      movel(pose_trans(ref_frame,p[0.079719, 0.078170, -0.000125, -0.013708, 3.141563, -0.000000]),accel_mss,speed_ms,0,0.001)
      movel(pose_trans(ref_frame,p[0.079740, 0.078322, -0.000125, -0.013708, 3.141563, 0.000000]),accel_mss,speed_ms,0,0.001)
      movel(pose_trans(ref_frame,p[0.079758, 0.078475, -0.000125, -0.013708, 3.141563, -0.000000]),accel_mss,speed_ms,0,0.001)
      movel(pose_trans(ref_frame,p[0.079771, 0.078603, -0.000125, -0.013708, 3.141563, 0.000000]),accel_mss,speed_ms,0,0.001)
      movel(pose_trans(ref_frame,p[0.079782, 0.078732, -0.000125, -0.013708, 3.141563, 0.000000]),accel_mss,speed_ms,0,0.001)
      movel(pose_trans(ref_frame,p[0.079779, 0.078758, -0.000125, -0.013708, 3.141563, 0.000000]),accel_mss,speed_ms,0,0.001)
      movel(pose_trans(ref_frame,p[0.079765, 0.078781, -0.000125, -0.013708, 3.141563, 0.000000]),accel_mss,speed_ms,0,0.001)
      movel(pose_trans(ref_frame,p[0.079742, 0.078796, -0.000125, -0.013708, 3.141563, 0.000000]),accel_mss,speed_ms,0,0.001)
      movel(pose_trans(ref_frame,p[0.079715, 0.078802, -0.000125, -0.013708, 3.141563, 0.000000]),accel_mss,speed_ms,0,0.001)
      movel(pose_trans(ref_frame,p[0.079591, 0.078803, -0.000125, -0.013708, 3.141563, 0.000000]),accel_mss,speed_ms,0,0.001)
      movel(pose_trans(ref_frame,p[0.079467, 0.078802, -0.000125, -0.013708, 3.141563, 0.000000]),accel_mss,speed_ms,0,0.001)
      movel(pose_trans(ref_frame,p[0.079319, 0.078800, -0.000125, -0.013708, 3.141563, -0.000000]),accel_mss,speed_ms,0,0.001)
      movel(pose_trans(ref_frame,p[0.079172, 0.078794, -0.000125, -0.013708, 3.141563, 0.000000]),accel_mss,speed_ms,0,0.001)
      movel(pose_trans(ref_frame,p[0.079002, 0.078785, -0.000125, -0.013708, 3.141563, 0.000000]),accel_mss,speed_ms,0,0.001)
      movel(pose_trans(ref_frame,p[0.078832, 0.078774, -0.000125, -0.013708, 3.141563, -0.000000]),accel_mss,speed_ms,0,0.001)
      movel(pose_trans(ref_frame,p[0.077770, 0.078748, -0.000125, -0.013708, 3.141563, -0.000000]),accel_mss,speed_ms,0,0.001)
      movel(pose_trans(ref_frame,p[0.076711, 0.078827, -0.000125, -0.013708, 3.141563, 0.000000]),accel_mss,speed_ms,0,0.001)
      movel(pose_trans(ref_frame,p[0.075653, 0.079010, -0.000125, -0.013708, 3.141563, -0.000000]),accel_mss,speed_ms,0,0.001)
      movel(pose_trans(ref_frame,p[0.074616, 0.079292, -0.000125, -0.013708, 3.141563, -0.000000]),accel_mss,speed_ms,0,0.001)
      movel(pose_trans(ref_frame,p[0.073606, 0.079674, -0.000125, -0.013708, 3.141563, 0.000000]),accel_mss,speed_ms,0,0.001)
      movel(pose_trans(ref_frame,p[0.072636, 0.080148, -0.000125, -0.013708, 3.141563, 0.000000]),accel_mss,speed_ms,0,0.001)
      movel(pose_trans(ref_frame,p[0.071716, 0.080712, -0.000125, -0.013708, 3.141563, -0.000000]),accel_mss,speed_ms,0,0.001)
      movel(pose_trans(ref_frame,p[0.070854, 0.081361, -0.000125, -0.013708, 3.141563, 0.000000]),accel_mss,speed_ms,0,0.001)
      movel(pose_trans(ref_frame,p[0.069464, 0.082689, -0.000125, -0.013708, 3.141563, 0.000000]),accel_mss,speed_ms,0,0.001)
      movel(pose_trans(ref_frame,p[0.068275, 0.084199, -0.000125, -0.013708, 3.141563, 0.000000]),accel_mss,speed_ms,0,0.001)
      movel(pose_trans(ref_frame,p[0.067302, 0.085869, -0.000125, -0.013708, 3.141563, -0.000000]),accel_mss,speed_ms,0,0.001)
      movel(pose_trans(ref_frame,p[0.066568, 0.087658, -0.000125, -0.013708, 3.141563, 0.000000]),accel_mss,speed_ms,0,0.001)
      movel(pose_trans(ref_frame,p[0.066058, 0.089620, -0.000125, -0.013708, 3.141563, 0.000000]),accel_mss,speed_ms,0,0.001)
      movel(pose_trans(ref_frame,p[0.065808, 0.091631, -0.000125, -0.013708, 3.141563, -0.000000]),accel_mss,speed_ms,0,0.001)
      movel(pose_trans(ref_frame,p[0.065796, 0.093809, -0.000125, -0.013708, 3.141563, 0.000000]),accel_mss,speed_ms,0,0.001)
      movel(pose_trans(ref_frame,p[0.066013, 0.095977, -0.000125, -0.013708, 3.141563, 0.000000]),accel_mss,speed_ms,0,0.001)
      movel(pose_trans(ref_frame,p[0.066187, 0.097070, -0.000125, -0.013708, 3.141563, 0.000000]),accel_mss,speed_ms,0,0.001)
      movel(pose_trans(ref_frame,p[0.066376, 0.098160, -0.000125, -0.013708, 3.141563, 0.000000]),accel_mss,speed_ms,0,0.001)
      movel(pose_trans(ref_frame,p[0.066549, 0.099068, -0.000125, -0.013708, 3.141563, -0.000000]),accel_mss,speed_ms,0,0.001)
      movel(pose_trans(ref_frame,p[0.066742, 0.099971, -0.000125, -0.013708, 3.141563, -0.000000]),accel_mss,speed_ms,0,0.001)
      movel(pose_trans(ref_frame,p[0.067000, 0.101082, -0.000125, -0.013708, 3.141563, 0.000000]),accel_mss,speed_ms,0,0.001)
      movel(pose_trans(ref_frame,p[0.067275, 0.102189, -0.000125, -0.013708, 3.141563, 0.000000]),accel_mss,speed_ms,0,0.001)
      movel(pose_trans(ref_frame,p[0.067780, 0.104154, -0.000125, -0.013708, 3.141563, 0.000000]),accel_mss,speed_ms,0,0.001)
      movel(pose_trans(ref_frame,p[0.068291, 0.106118, -0.000125, -0.013708, 3.141563, 0.000000]),accel_mss,speed_ms,0,0.001)
      movel(pose_trans(ref_frame,p[0.068671, 0.107644, -0.000125, -0.013708, 3.141563, 0.000000]),accel_mss,speed_ms,0,0.001)
      movel(pose_trans(ref_frame,p[0.069013, 0.109180, -0.000125, -0.013708, 3.141563, 0.000000]),accel_mss,speed_ms,0,0.001)
      movel(pose_trans(ref_frame,p[0.069211, 0.110301, -0.000125, -0.013708, 3.141563, -0.000000]),accel_mss,speed_ms,0,0.001)
      movel(pose_trans(ref_frame,p[0.069339, 0.111433, -0.000125, -0.013708, 3.141563, 0.000000]),accel_mss,speed_ms,0,0.001)
      movel(pose_trans(ref_frame,p[0.069369, 0.112274, -0.000125, -0.013708, 3.141563, 0.000000]),accel_mss,speed_ms,0,0.001)
      movel(pose_trans(ref_frame,p[0.069325, 0.113114, -0.000125, -0.013708, 3.141563, -0.000000]),accel_mss,speed_ms,0,0.001)
      movel(pose_trans(ref_frame,p[0.069201, 0.113740, -0.000125, -0.013708, 3.141563, 0.000000]),accel_mss,speed_ms,0,0.001)
      movel(pose_trans(ref_frame,p[0.068955, 0.114330, -0.000125, -0.013708, 3.141563, -0.000000]),accel_mss,speed_ms,0,0.001)
      movel(pose_trans(ref_frame,p[0.068717, 0.114661, -0.000125, -0.013708, 3.141563, -0.000000]),accel_mss,speed_ms,0,0.001)
      movel(pose_trans(ref_frame,p[0.068403, 0.114922, -0.000125, -0.013708, 3.141563, -0.000000]),accel_mss,speed_ms,0,0.001)
      movel(pose_trans(ref_frame,p[0.068014, 0.115112, -0.000125, -0.013708, 3.141563, -0.000000]),accel_mss,speed_ms,0,0.001)
      movel(pose_trans(ref_frame,p[0.067594, 0.115214, -0.000125, -0.013708, 3.141563, 0.000000]),accel_mss,speed_ms,0,0.001)
      movel(pose_trans(ref_frame,p[0.067102, 0.115233, -0.000125, -0.013708, 3.141563, 0.000000]),accel_mss,speed_ms,0,0.001)
      movel(pose_trans(ref_frame,p[0.066615, 0.115163, -0.000125, -0.013708, 3.141563, 0.000000]),accel_mss,speed_ms,0,0.001)
      movel(pose_trans(ref_frame,p[0.066086, 0.115001, -0.000125, -0.013708, 3.141563, 0.000000]),accel_mss,speed_ms,0,0.001)
      movel(pose_trans(ref_frame,p[0.065582, 0.114772, -0.000125, -0.013708, 3.141563, -0.000000]),accel_mss,speed_ms,0,0.001)
      movel(pose_trans(ref_frame,p[0.065310, 0.114617, -0.000125, -0.013708, 3.141563, 0.000000]),accel_mss,speed_ms,0,0.001)
      movel(pose_trans(ref_frame,p[0.065046, 0.114448, -0.000125, -0.013708, 3.141563, 0.000000]),accel_mss,speed_ms,0,0.001)
      movel(pose_trans(ref_frame,p[0.064814, 0.114277, -0.000125, -0.013708, 3.141563, 0.000000]),accel_mss,speed_ms,0,0.001)
      movel(pose_trans(ref_frame,p[0.064595, 0.114091, -0.000125, -0.013708, 3.141563, 0.000000]),accel_mss,speed_ms,0,0.001)
      movel(pose_trans(ref_frame,p[0.064291, 0.113805, -0.000125, -0.013708, 3.141563, -0.000000]),accel_mss,speed_ms,0,0.001)
      movel(pose_trans(ref_frame,p[0.063997, 0.113510, -0.000125, -0.013708, 3.141563, -0.000000]),accel_mss,speed_ms,0,0.001)
      movel(pose_trans(ref_frame,p[0.063336, 0.112821, -0.000125, -0.013708, 3.141563, -0.000000]),accel_mss,speed_ms,0,0.001)
      movel(pose_trans(ref_frame,p[0.062678, 0.112129, -0.000125, -0.013708, 3.141563, 0.000000]),accel_mss,speed_ms,0,0.001)
      movel(pose_trans(ref_frame,p[0.062101, 0.111524, -0.000125, -0.013708, 3.141563, 0.000000]),accel_mss,speed_ms,0,0.001)
      movel(pose_trans(ref_frame,p[0.061522, 0.110923, -0.000125, -0.013708, 3.141563, 0.000000]),accel_mss,speed_ms,0,0.001)
      movel(pose_trans(ref_frame,p[0.061175, 0.110572, -0.000125, -0.013708, 3.141563, -0.000000]),accel_mss,speed_ms,0,0.001)
      movel(pose_trans(ref_frame,p[0.060820, 0.110229, -0.000125, -0.013708, 3.141563, -0.000000]),accel_mss,speed_ms,0,0.001)
      movel(pose_trans(ref_frame,p[0.060559, 0.109992, -0.000125, -0.013708, 3.141563, 0.000000]),accel_mss,speed_ms,0,0.001)
      movel(pose_trans(ref_frame,p[0.060290, 0.109764, -0.000125, -0.013708, 3.141563, 0.000000]),accel_mss,speed_ms,0,0.001)
      movel(pose_trans(ref_frame,p[0.060039, 0.109570, -0.000125, -0.013708, 3.141563, 0.000000]),accel_mss,speed_ms,0,0.001)
      movel(pose_trans(ref_frame,p[0.059778, 0.109389, -0.000125, -0.013708, 3.141563, 0.000000]),accel_mss,speed_ms,0,0.001)
      movel(pose_trans(ref_frame,p[0.059074, 0.108952, -0.000125, -0.013708, 3.141563, 0.000000]),accel_mss,speed_ms,0,0.001)
      movel(pose_trans(ref_frame,p[0.058348, 0.108551, -0.000125, -0.013708, 3.141563, -0.000000]),accel_mss,speed_ms,0,0.001)
      movel(pose_trans(ref_frame,p[0.057513, 0.108137, -0.000125, -0.013708, 3.141563, -0.000000]),accel_mss,speed_ms,0,0.001)
      movel(pose_trans(ref_frame,p[0.056662, 0.107753, -0.000125, -0.013708, 3.141563, 0.000000]),accel_mss,speed_ms,0,0.001)
      movel(pose_trans(ref_frame,p[0.055839, 0.107417, -0.000125, -0.013708, 3.141563, 0.000000]),accel_mss,speed_ms,0,0.001)
      movel(pose_trans(ref_frame,p[0.055003, 0.107111, -0.000125, -0.013708, 3.141563, -0.000000]),accel_mss,speed_ms,0,0.001)
      movel(pose_trans(ref_frame,p[0.054348, 0.106914, -0.000125, -0.013708, 3.141563, -0.000000]),accel_mss,speed_ms,0,0.001)
      movel(pose_trans(ref_frame,p[0.053678, 0.106769, -0.000125, -0.013708, 3.141563, -0.000000]),accel_mss,speed_ms,0,0.001)
      movel(pose_trans(ref_frame,p[0.053472, 0.106738, -0.000125, -0.013708, 3.141563, -0.000000]),accel_mss,speed_ms,0,0.001)
      movel(pose_trans(ref_frame,p[0.053265, 0.106717, -0.000125, -0.013708, 3.141563, 0.000000]),accel_mss,speed_ms,0,0.001)
      movel(pose_trans(ref_frame,p[0.052975, 0.106698, -0.000125, -0.013708, 3.141563, -0.000000]),accel_mss,speed_ms,0,0.001)
      movel(pose_trans(ref_frame,p[0.052685, 0.106684, -0.000125, -0.013708, 3.141563, -0.000000]),accel_mss,speed_ms,0,0.001)
      movel(pose_trans(ref_frame,p[0.052370, 0.106675, -0.000125, -0.013708, 3.141563, 0.000000]),accel_mss,speed_ms,0,0.001)
      movel(pose_trans(ref_frame,p[0.052053, 0.106672, -0.000125, -0.013708, 3.141563, 0.000000]),accel_mss,speed_ms,0,0.001)
      movel(pose_trans(ref_frame,p[0.051757, 0.106675, -0.000125, -0.013708, 3.141563, 0.000000]),accel_mss,speed_ms,0,0.001)
      movel(pose_trans(ref_frame,p[0.051461, 0.106685, -0.000125, -0.013708, 3.141563, 0.000000]),accel_mss,speed_ms,0,0.001)
      movel(pose_trans(ref_frame,p[0.050758, 0.106709, -0.000125, -0.013708, 3.141563, 0.000000]),accel_mss,speed_ms,0,0.001)
      movel(pose_trans(ref_frame,p[0.050054, 0.106718, -0.000125, -0.013708, 3.141563, -0.000000]),accel_mss,speed_ms,0,0.001)
      movel(pose_trans(ref_frame,p[0.049710, 0.106695, -0.000125, -0.013708, 3.141563, 0.000000]),accel_mss,speed_ms,0,0.001)
      movel(pose_trans(ref_frame,p[0.049372, 0.106623, -0.000125, -0.013708, 3.141563, -0.000000]),accel_mss,speed_ms,0,0.001)
      movel(pose_trans(ref_frame,p[0.049067, 0.106508, -0.000125, -0.013708, 3.141563, 0.000000]),accel_mss,speed_ms,0,0.001)
      movel(pose_trans(ref_frame,p[0.048785, 0.106344, -0.000125, -0.013708, 3.141563, 0.000000]),accel_mss,speed_ms,0,0.001)
      movel(pose_trans(ref_frame,p[0.048308, 0.106001, -0.000125, -0.013708, 3.141563, 0.000000]),accel_mss,speed_ms,0,0.001)
      movel(pose_trans(ref_frame,p[0.047842, 0.105642, -0.000125, -0.013708, 3.141563, -0.000000]),accel_mss,speed_ms,0,0.001)
      movel(pose_trans(ref_frame,p[0.047407, 0.105304, -0.000125, -0.013708, 3.141563, -0.000000]),accel_mss,speed_ms,0,0.001)
      movel(pose_trans(ref_frame,p[0.046966, 0.104974, -0.000125, -0.013708, 3.141563, -0.000000]),accel_mss,speed_ms,0,0.001)
      movel(pose_trans(ref_frame,p[0.046600, 0.104716, -0.000125, -0.013708, 3.141563, 0.000000]),accel_mss,speed_ms,0,0.001)
      movel(pose_trans(ref_frame,p[0.046224, 0.104471, -0.000125, -0.013708, 3.141563, -0.000000]),accel_mss,speed_ms,0,0.001)
      movel(pose_trans(ref_frame,p[0.045908, 0.104283, -0.000125, -0.013708, 3.141563, 0.000000]),accel_mss,speed_ms,0,0.001)
      movel(pose_trans(ref_frame,p[0.045584, 0.104109, -0.000125, -0.013708, 3.141563, -0.000000]),accel_mss,speed_ms,0,0.001)
      movel(pose_trans(ref_frame,p[0.045312, 0.103984, -0.000125, -0.013708, 3.141563, 0.000000]),accel_mss,speed_ms,0,0.001)
      movel(pose_trans(ref_frame,p[0.045030, 0.103881, -0.000125, -0.013708, 3.141563, 0.000000]),accel_mss,speed_ms,0,0.001)
      movel(pose_trans(ref_frame,p[0.044911, 0.103850, -0.000125, -0.013708, 3.141563, 0.000000]),accel_mss,speed_ms,0,0.001)
      movel(pose_trans(ref_frame,p[0.044789, 0.103833, -0.000125, -0.013708, 3.141563, 0.000000]),accel_mss,speed_ms,0,0.001)
      movel(pose_trans(ref_frame,p[0.044526, 0.103812, -0.000125, -0.013708, 3.141563, -0.000000]),accel_mss,speed_ms,0,0.001)
      movel(pose_trans(ref_frame,p[0.044263, 0.103794, -0.000125, -0.013708, 3.141563, 0.000000]),accel_mss,speed_ms,0,0.001)
      movel(pose_trans(ref_frame,p[0.043949, 0.103779, -0.000125, -0.013708, 3.141563, 0.000000]),accel_mss,speed_ms,0,0.001)
      movel(pose_trans(ref_frame,p[0.043635, 0.103769, -0.000125, -0.013708, 3.141563, -0.000000]),accel_mss,speed_ms,0,0.001)
      movel(pose_trans(ref_frame,p[0.043300, 0.103763, -0.000125, -0.013708, 3.141563, -0.000000]),accel_mss,speed_ms,0,0.001)
      movel(pose_trans(ref_frame,p[0.042965, 0.103761, -0.000125, -0.013708, 3.141563, 0.000000]),accel_mss,speed_ms,0,0.001)
      movel(pose_trans(ref_frame,p[0.042438, 0.103756, -0.000125, -0.013708, 3.141563, -0.000000]),accel_mss,speed_ms,0,0.001)
      movel(pose_trans(ref_frame,p[0.041911, 0.103737, -0.000125, -0.013708, 3.141563, 0.000000]),accel_mss,speed_ms,0,0.001)
      movel(pose_trans(ref_frame,p[0.041500, 0.103706, -0.000125, -0.013708, 3.141563, 0.000000]),accel_mss,speed_ms,0,0.001)
      movel(pose_trans(ref_frame,p[0.041092, 0.103653, -0.000125, -0.013708, 3.141563, 0.000000]),accel_mss,speed_ms,0,0.001)
      movel(pose_trans(ref_frame,p[0.040790, 0.103594, -0.000125, -0.013708, 3.141563, -0.000000]),accel_mss,speed_ms,0,0.001)
      movel(pose_trans(ref_frame,p[0.040491, 0.103516, -0.000125, -0.013708, 3.141563, 0.000000]),accel_mss,speed_ms,0,0.001)
      movel(pose_trans(ref_frame,p[0.040314, 0.103437, -0.000125, -0.013708, 3.141563, 0.000000]),accel_mss,speed_ms,0,0.001)
      movel(pose_trans(ref_frame,p[0.040160, 0.103318, -0.000125, -0.013708, 3.141563, -0.000000]),accel_mss,speed_ms,0,0.001)
      movel(pose_trans(ref_frame,p[0.040130, 0.103293, -0.000125, -0.013708, 3.141563, 0.000000]),accel_mss,speed_ms,0,0.001)
      movel(pose_trans(ref_frame,p[0.040097, 0.103273, -0.000125, -0.013708, 3.141563, 0.000000]),accel_mss,speed_ms,0,0.001)
      movel(pose_trans(ref_frame,p[0.040052, 0.103254, -0.000125, -0.013708, 3.141563, -0.000000]),accel_mss,speed_ms,0,0.001)
      movel(pose_trans(ref_frame,p[0.040006, 0.103239, -0.000125, -0.013708, 3.141563, 0.000000]),accel_mss,speed_ms,0,0.001)
      movel(pose_trans(ref_frame,p[0.039955, 0.103227, -0.000125, -0.013708, 3.141563, -0.000000]),accel_mss,speed_ms,0,0.001)
      movel(pose_trans(ref_frame,p[0.039904, 0.103220, -0.000125, -0.013708, 3.141563, -0.000000]),accel_mss,speed_ms,0,0.001)
      movel(pose_trans(ref_frame,p[0.039855, 0.103217, -0.000125, -0.013708, 3.141563, 0.000000]),accel_mss,speed_ms,0,0.001)
      movel(pose_trans(ref_frame,p[0.039805, 0.103219, -0.000125, -0.013708, 3.141563, -0.000000]),accel_mss,speed_ms,0,0.001)
      movel(pose_trans(ref_frame,p[0.039745, 0.103228, -0.000125, -0.013708, 3.141563, 0.000000]),accel_mss,speed_ms,0,0.001)
      movel(pose_trans(ref_frame,p[0.039686, 0.103242, -0.000125, -0.013708, 3.141563, -0.000000]),accel_mss,speed_ms,0,0.001)
      movel(pose_trans(ref_frame,p[0.039647, 0.103260, -0.000125, -0.013708, 3.141563, -0.000000]),accel_mss,speed_ms,0,0.001)
      movel(pose_trans(ref_frame,p[0.039613, 0.103287, -0.000125, -0.013708, 3.141563, 0.000000]),accel_mss,speed_ms,0,0.001)
      movel(pose_trans(ref_frame,p[0.039587, 0.103323, -0.000125, -0.013708, 3.141563, 0.000000]),accel_mss,speed_ms,0,0.001)
      movel(pose_trans(ref_frame,p[0.039571, 0.103364, -0.000125, -0.013708, 3.141563, 0.000000]),accel_mss,speed_ms,0,0.001)
      movel(pose_trans(ref_frame,p[0.039557, 0.103428, -0.000125, -0.013708, 3.141563, -0.000000]),accel_mss,speed_ms,0,0.001)
      movel(pose_trans(ref_frame,p[0.039548, 0.103493, -0.000125, -0.013708, 3.141563, 0.000000]),accel_mss,speed_ms,0,0.001)
      movel(pose_trans(ref_frame,p[0.039567, 0.103662, -0.000125, -0.013708, 3.141563, 0.000000]),accel_mss,speed_ms,0,0.001)
      movel(pose_trans(ref_frame,p[0.039653, 0.103808, -0.000125, -0.013708, 3.141563, -0.000000]),accel_mss,speed_ms,0,0.001)
      movel(pose_trans(ref_frame,p[0.039898, 0.104063, -0.000125, -0.013708, 3.141563, 0.000000]),accel_mss,speed_ms,0,0.001)
      movel(pose_trans(ref_frame,p[0.040158, 0.104302, -0.000125, -0.013708, 3.141563, -0.000000]),accel_mss,speed_ms,0,0.001)
      movel(pose_trans(ref_frame,p[0.040460, 0.104548, -0.000125, -0.013708, 3.141563, 0.000000]),accel_mss,speed_ms,0,0.001)
      movel(pose_trans(ref_frame,p[0.040778, 0.104773, -0.000125, -0.013708, 3.141563, 0.000000]),accel_mss,speed_ms,0,0.001)
      movel(pose_trans(ref_frame,p[0.041066, 0.104942, -0.000125, -0.013708, 3.141563, 0.000000]),accel_mss,speed_ms,0,0.001)
      movel(pose_trans(ref_frame,p[0.041370, 0.105079, -0.000125, -0.013708, 3.141563, 0.000000]),accel_mss,speed_ms,0,0) # end trace
      speed_ms    = 1.000
      movel(pose_trans(ref_frame,p[0.041370, 0.105079, 0.005000, -0.013708, 3.141563, 0.000000]),accel_mss,speed_ms,0,0.001)
      movel(pose_trans(ref_frame,p[0.055107, 0.114922, 0.005000, -0.013708, 3.141563, 0.000000]),accel_mss,speed_ms,0,0) # end trace
      speed_ms    = 0.002
      movel(pose_trans(ref_frame,p[0.055107, 0.114922, -0.000125, -0.013708, 3.141563, 0.000000]),accel_mss,speed_ms,0,0) # end trace
      speed_ms    = 0.007
      movel(pose_trans(ref_frame,p[0.055327, 0.115016, -0.000125, -0.013708, 3.141563, -0.000000]),accel_mss,speed_ms,0,0.001)
      movel(pose_trans(ref_frame,p[0.055556, 0.115086, -0.000125, -0.013708, 3.141563, -0.000000]),accel_mss,speed_ms,0,0.001)
      movel(pose_trans(ref_frame,p[0.055772, 0.115124, -0.000125, -0.013708, 3.141563, -0.000000]),accel_mss,speed_ms,0,0.001)
      movel(pose_trans(ref_frame,p[0.055992, 0.115132, -0.000125, -0.013708, 3.141563, 0.000000]),accel_mss,speed_ms,0,0.001)
      movel(pose_trans(ref_frame,p[0.056174, 0.115110, -0.000125, -0.013708, 3.141563, 0.000000]),accel_mss,speed_ms,0,0.001)
      movel(pose_trans(ref_frame,p[0.056349, 0.115058, -0.000125, -0.013708, 3.141563, -0.000000]),accel_mss,speed_ms,0,0.001)
      movel(pose_trans(ref_frame,p[0.056474, 0.114984, -0.000125, -0.013708, 3.141563, -0.000000]),accel_mss,speed_ms,0,0.001)
      movel(pose_trans(ref_frame,p[0.056569, 0.114873, -0.000125, -0.013708, 3.141563, -0.000000]),accel_mss,speed_ms,0,0.001)
      movel(pose_trans(ref_frame,p[0.056614, 0.114817, -0.000125, -0.013708, 3.141563, -0.000000]),accel_mss,speed_ms,0,0.001)
      movel(pose_trans(ref_frame,p[0.056671, 0.114776, -0.000125, -0.013708, 3.141563, 0.000000]),accel_mss,speed_ms,0,0.001)
      movel(pose_trans(ref_frame,p[0.056741, 0.114748, -0.000125, -0.013708, 3.141563, 0.000000]),accel_mss,speed_ms,0,0.001)
      movel(pose_trans(ref_frame,p[0.056815, 0.114736, -0.000125, -0.013708, 3.141563, 0.000000]),accel_mss,speed_ms,0,0.001)
      movel(pose_trans(ref_frame,p[0.056926, 0.114738, -0.000125, -0.013708, 3.141563, -0.000000]),accel_mss,speed_ms,0,0.001)
      movel(pose_trans(ref_frame,p[0.057036, 0.114754, -0.000125, -0.013708, 3.141563, 0.000000]),accel_mss,speed_ms,0,0.001)
      movel(pose_trans(ref_frame,p[0.057220, 0.114794, -0.000125, -0.013708, 3.141563, 0.000000]),accel_mss,speed_ms,0,0.001)
      movel(pose_trans(ref_frame,p[0.057403, 0.114839, -0.000125, -0.013708, 3.141563, 0.000000]),accel_mss,speed_ms,0,0.001)
      movel(pose_trans(ref_frame,p[0.057700, 0.114903, -0.000125, -0.013708, 3.141563, 0.000000]),accel_mss,speed_ms,0,0.001)
      movel(pose_trans(ref_frame,p[0.058001, 0.114941, -0.000125, -0.013708, 3.141563, 0.000000]),accel_mss,speed_ms,0,0.001)
      movel(pose_trans(ref_frame,p[0.058171, 0.114920, -0.000125, -0.013708, 3.141563, 0.000000]),accel_mss,speed_ms,0,0.001)
      movel(pose_trans(ref_frame,p[0.058318, 0.114832, -0.000125, -0.013708, 3.141563, 0.000000]),accel_mss,speed_ms,0,0.001)
      movel(pose_trans(ref_frame,p[0.058413, 0.114693, -0.000125, -0.013708, 3.141563, 0.000000]),accel_mss,speed_ms,0,0.001)
      movel(pose_trans(ref_frame,p[0.058442, 0.114528, -0.000125, -0.013708, 3.141563, 0.000000]),accel_mss,speed_ms,0,0.001)
      movel(pose_trans(ref_frame,p[0.058415, 0.114235, -0.000125, -0.013708, 3.141563, -0.000000]),accel_mss,speed_ms,0,0.001)
      movel(pose_trans(ref_frame,p[0.058361, 0.113947, -0.000125, -0.013708, 3.141563, -0.000000]),accel_mss,speed_ms,0,0.001)
      movel(pose_trans(ref_frame,p[0.058310, 0.113755, -0.000125, -0.013708, 3.141563, -0.000000]),accel_mss,speed_ms,0,0.001)
      movel(pose_trans(ref_frame,p[0.058249, 0.113567, -0.000125, -0.013708, 3.141563, -0.000000]),accel_mss,speed_ms,0,0.001)
      movel(pose_trans(ref_frame,p[0.058187, 0.113415, -0.000125, -0.013708, 3.141563, 0.000000]),accel_mss,speed_ms,0,0.001)
      movel(pose_trans(ref_frame,p[0.058111, 0.113269, -0.000125, -0.013708, 3.141563, 0.000000]),accel_mss,speed_ms,0,0.001)
      movel(pose_trans(ref_frame,p[0.058011, 0.113113, -0.000125, -0.013708, 3.141563, -0.000000]),accel_mss,speed_ms,0,0.001)
      movel(pose_trans(ref_frame,p[0.057900, 0.112965, -0.000125, -0.013708, 3.141563, -0.000000]),accel_mss,speed_ms,0,0.001)
      movel(pose_trans(ref_frame,p[0.057722, 0.112753, -0.000125, -0.013708, 3.141563, -0.000000]),accel_mss,speed_ms,0,0.001)
      movel(pose_trans(ref_frame,p[0.057540, 0.112545, -0.000125, -0.013708, 3.141563, 0.000000]),accel_mss,speed_ms,0,0.001)
      movel(pose_trans(ref_frame,p[0.057372, 0.112362, -0.000125, -0.013708, 3.141563, -0.000000]),accel_mss,speed_ms,0,0.001)
      movel(pose_trans(ref_frame,p[0.057201, 0.112181, -0.000125, -0.013708, 3.141563, -0.000000]),accel_mss,speed_ms,0,0.001)
      movel(pose_trans(ref_frame,p[0.057089, 0.112072, -0.000125, -0.013708, 3.141563, 0.000000]),accel_mss,speed_ms,0,0.001)
      movel(pose_trans(ref_frame,p[0.056971, 0.111969, -0.000125, -0.013708, 3.141563, -0.000000]),accel_mss,speed_ms,0,0.001)
      movel(pose_trans(ref_frame,p[0.056886, 0.111908, -0.000125, -0.013708, 3.141563, -0.000000]),accel_mss,speed_ms,0,0.001)
      movel(pose_trans(ref_frame,p[0.056796, 0.111855, -0.000125, -0.013708, 3.141563, 0.000000]),accel_mss,speed_ms,0,0.001)
      movel(pose_trans(ref_frame,p[0.056728, 0.111831, -0.000125, -0.013708, 3.141563, 0.000000]),accel_mss,speed_ms,0,0.001)
      movel(pose_trans(ref_frame,p[0.056655, 0.111828, -0.000125, -0.013708, 3.141563, 0.000000]),accel_mss,speed_ms,0,0.001)
      movel(pose_trans(ref_frame,p[0.056545, 0.111854, -0.000125, -0.013708, 3.141563, 0.000000]),accel_mss,speed_ms,0,0.001)
      movel(pose_trans(ref_frame,p[0.056447, 0.111910, -0.000125, -0.013708, 3.141563, 0.000000]),accel_mss,speed_ms,0,0.001)
      movel(pose_trans(ref_frame,p[0.056363, 0.111995, -0.000125, -0.013708, 3.141563, -0.000000]),accel_mss,speed_ms,0,0.001)
      movel(pose_trans(ref_frame,p[0.056302, 0.112097, -0.000125, -0.013708, 3.141563, 0.000000]),accel_mss,speed_ms,0,0.001)
      movel(pose_trans(ref_frame,p[0.056259, 0.112229, -0.000125, -0.013708, 3.141563, 0.000000]),accel_mss,speed_ms,0,0.001)
      movel(pose_trans(ref_frame,p[0.056244, 0.112366, -0.000125, -0.013708, 3.141563, -0.000000]),accel_mss,speed_ms,0,0.001)
      movel(pose_trans(ref_frame,p[0.056252, 0.112525, -0.000125, -0.013708, 3.141563, 0.000000]),accel_mss,speed_ms,0,0.001)
      movel(pose_trans(ref_frame,p[0.056281, 0.112681, -0.000125, -0.013708, 3.141563, 0.000000]),accel_mss,speed_ms,0,0.001)
      movel(pose_trans(ref_frame,p[0.056303, 0.112785, -0.000125, -0.013708, 3.141563, 0.000000]),accel_mss,speed_ms,0,0.001)
      movel(pose_trans(ref_frame,p[0.056318, 0.112890, -0.000125, -0.013708, 3.141563, 0.000000]),accel_mss,speed_ms,0,0.001)
      movel(pose_trans(ref_frame,p[0.056318, 0.112972, -0.000125, -0.013708, 3.141563, 0.000000]),accel_mss,speed_ms,0,0.001)
      movel(pose_trans(ref_frame,p[0.056305, 0.113052, -0.000125, -0.013708, 3.141563, -0.000000]),accel_mss,speed_ms,0,0.001)
      movel(pose_trans(ref_frame,p[0.056278, 0.113127, -0.000125, -0.013708, 3.141563, -0.000000]),accel_mss,speed_ms,0,0.001)
      movel(pose_trans(ref_frame,p[0.056239, 0.113196, -0.000125, -0.013708, 3.141563, 0.000000]),accel_mss,speed_ms,0,0.001)
      movel(pose_trans(ref_frame,p[0.056178, 0.113276, -0.000125, -0.013708, 3.141563, -0.000000]),accel_mss,speed_ms,0,0.001)
      movel(pose_trans(ref_frame,p[0.056110, 0.113350, -0.000125, -0.013708, 3.141563, 0.000000]),accel_mss,speed_ms,0,0.001)
      movel(pose_trans(ref_frame,p[0.055933, 0.113516, -0.000125, -0.013708, 3.141563, -0.000000]),accel_mss,speed_ms,0,0.001)
      movel(pose_trans(ref_frame,p[0.055749, 0.113675, -0.000125, -0.013708, 3.141563, 0.000000]),accel_mss,speed_ms,0,0.001)
      movel(pose_trans(ref_frame,p[0.055632, 0.113750, -0.000125, -0.013708, 3.141563, -0.000000]),accel_mss,speed_ms,0,0.001)
      movel(pose_trans(ref_frame,p[0.055502, 0.113798, -0.000125, -0.013708, 3.141563, 0.000000]),accel_mss,speed_ms,0,0.001)
      movel(pose_trans(ref_frame,p[0.055392, 0.113804, -0.000125, -0.013708, 3.141563, 0.000000]),accel_mss,speed_ms,0,0.001)
      movel(pose_trans(ref_frame,p[0.055286, 0.113773, -0.000125, -0.013708, 3.141563, 0.000000]),accel_mss,speed_ms,0,0.001)
      movel(pose_trans(ref_frame,p[0.055163, 0.113698, -0.000125, -0.013708, 3.141563, 0.000000]),accel_mss,speed_ms,0,0.001)
      movel(pose_trans(ref_frame,p[0.055053, 0.113605, -0.000125, -0.013708, 3.141563, 0.000000]),accel_mss,speed_ms,0,0.001)
      movel(pose_trans(ref_frame,p[0.054907, 0.113440, -0.000125, -0.013708, 3.141563, -0.000000]),accel_mss,speed_ms,0,0.001)
      movel(pose_trans(ref_frame,p[0.054782, 0.113260, -0.000125, -0.013708, 3.141563, 0.000000]),accel_mss,speed_ms,0,0.001)
      movel(pose_trans(ref_frame,p[0.054680, 0.113064, -0.000125, -0.013708, 3.141563, 0.000000]),accel_mss,speed_ms,0,0.001)
      movel(pose_trans(ref_frame,p[0.054601, 0.112858, -0.000125, -0.013708, 3.141563, -0.000000]),accel_mss,speed_ms,0,0.001)
      movel(pose_trans(ref_frame,p[0.054555, 0.112670, -0.000125, -0.013708, 3.141563, 0.000000]),accel_mss,speed_ms,0,0.001)
      movel(pose_trans(ref_frame,p[0.054535, 0.112479, -0.000125, -0.013708, 3.141563, 0.000000]),accel_mss,speed_ms,0,0.001)
      movel(pose_trans(ref_frame,p[0.054552, 0.112336, -0.000125, -0.013708, 3.141563, 0.000000]),accel_mss,speed_ms,0,0.001)
      movel(pose_trans(ref_frame,p[0.054611, 0.112205, -0.000125, -0.013708, 3.141563, 0.000000]),accel_mss,speed_ms,0,0.001)
      movel(pose_trans(ref_frame,p[0.054648, 0.112149, -0.000125, -0.013708, 3.141563, 0.000000]),accel_mss,speed_ms,0,0.001)
      movel(pose_trans(ref_frame,p[0.054685, 0.112093, -0.000125, -0.013708, 3.141563, 0.000000]),accel_mss,speed_ms,0,0.001)
      movel(pose_trans(ref_frame,p[0.054730, 0.112024, -0.000125, -0.013708, 3.141563, 0.000000]),accel_mss,speed_ms,0,0.001)
      movel(pose_trans(ref_frame,p[0.054775, 0.111956, -0.000125, -0.013708, 3.141563, -0.000000]),accel_mss,speed_ms,0,0.001)
      movel(pose_trans(ref_frame,p[0.054820, 0.111888, -0.000125, -0.013708, 3.141563, 0.000000]),accel_mss,speed_ms,0,0.001)
      movel(pose_trans(ref_frame,p[0.054865, 0.111819, -0.000125, -0.013708, 3.141563, 0.000000]),accel_mss,speed_ms,0,0.001)
      movel(pose_trans(ref_frame,p[0.054903, 0.111761, -0.000125, -0.013708, 3.141563, -0.000000]),accel_mss,speed_ms,0,0.001)
      movel(pose_trans(ref_frame,p[0.054941, 0.111703, -0.000125, -0.013708, 3.141563, 0.000000]),accel_mss,speed_ms,0,0.001)
      movel(pose_trans(ref_frame,p[0.054994, 0.111593, -0.000125, -0.013708, 3.141563, 0.000000]),accel_mss,speed_ms,0,0.001)
      movel(pose_trans(ref_frame,p[0.055014, 0.111473, -0.000125, -0.013708, 3.141563, 0.000000]),accel_mss,speed_ms,0,0.001)
      movel(pose_trans(ref_frame,p[0.054995, 0.111371, -0.000125, -0.013708, 3.141563, 0.000000]),accel_mss,speed_ms,0,0.001)
      movel(pose_trans(ref_frame,p[0.054935, 0.111286, -0.000125, -0.013708, 3.141563, -0.000000]),accel_mss,speed_ms,0,0.001)
      movel(pose_trans(ref_frame,p[0.054814, 0.111199, -0.000125, -0.013708, 3.141563, -0.000000]),accel_mss,speed_ms,0,0.001)
      movel(pose_trans(ref_frame,p[0.054676, 0.111142, -0.000125, -0.013708, 3.141563, 0.000000]),accel_mss,speed_ms,0,0.001)
      movel(pose_trans(ref_frame,p[0.054444, 0.111083, -0.000125, -0.013708, 3.141563, 0.000000]),accel_mss,speed_ms,0,0.001)
      movel(pose_trans(ref_frame,p[0.054209, 0.111039, -0.000125, -0.013708, 3.141563, 0.000000]),accel_mss,speed_ms,0,0.001)
      movel(pose_trans(ref_frame,p[0.053886, 0.111012, -0.000125, -0.013708, 3.141563, -0.000000]),accel_mss,speed_ms,0,0.001)
      movel(pose_trans(ref_frame,p[0.053563, 0.111036, -0.000125, -0.013708, 3.141563, 0.000000]),accel_mss,speed_ms,0,0.001)
      movel(pose_trans(ref_frame,p[0.053349, 0.111116, -0.000125, -0.013708, 3.141563, 0.000000]),accel_mss,speed_ms,0,0.001)
      movel(pose_trans(ref_frame,p[0.053184, 0.111275, -0.000125, -0.013708, 3.141563, 0.000000]),accel_mss,speed_ms,0,0.001)
      movel(pose_trans(ref_frame,p[0.053082, 0.111503, -0.000125, -0.013708, 3.141563, -0.000000]),accel_mss,speed_ms,0,0.001)
      movel(pose_trans(ref_frame,p[0.053063, 0.111752, -0.000125, -0.013708, 3.141563, 0.000000]),accel_mss,speed_ms,0,0.001)
      movel(pose_trans(ref_frame,p[0.053123, 0.112125, -0.000125, -0.013708, 3.141563, -0.000000]),accel_mss,speed_ms,0,0.001)
      movel(pose_trans(ref_frame,p[0.053222, 0.112490, -0.000125, -0.013708, 3.141563, -0.000000]),accel_mss,speed_ms,0,0.001)
      movel(pose_trans(ref_frame,p[0.053379, 0.112916, -0.000125, -0.013708, 3.141563, 0.000000]),accel_mss,speed_ms,0,0.001)
      movel(pose_trans(ref_frame,p[0.053565, 0.113330, -0.000125, -0.013708, 3.141563, 0.000000]),accel_mss,speed_ms,0,0.001)
      movel(pose_trans(ref_frame,p[0.053759, 0.113678, -0.000125, -0.013708, 3.141563, 0.000000]),accel_mss,speed_ms,0,0.001)
      movel(pose_trans(ref_frame,p[0.053986, 0.114004, -0.000125, -0.013708, 3.141563, -0.000000]),accel_mss,speed_ms,0,0.001)
      movel(pose_trans(ref_frame,p[0.054227, 0.114281, -0.000125, -0.013708, 3.141563, -0.000000]),accel_mss,speed_ms,0,0.001)
      movel(pose_trans(ref_frame,p[0.054496, 0.114529, -0.000125, -0.013708, 3.141563, -0.000000]),accel_mss,speed_ms,0,0.001)
      movel(pose_trans(ref_frame,p[0.054790, 0.114743, -0.000125, -0.013708, 3.141563, -0.000000]),accel_mss,speed_ms,0,0.001)
      movel(pose_trans(ref_frame,p[0.055107, 0.114922, -0.000125, -0.013708, 3.141563, 0.000000]),accel_mss,speed_ms,0,0) # end trace
      speed_ms    = 1.000
      movel(pose_trans(ref_frame,p[0.055107, 0.114922, 0.005000, -0.013708, 3.141563, 0.000000]),accel_mss,speed_ms,0,0.001)
      movel(pose_trans(ref_frame,p[0.077984, 0.140117, 0.005000, -0.013708, 3.141563, 0.000000]),accel_mss,speed_ms,0,0) # end trace
      speed_ms    = 0.002
      movel(pose_trans(ref_frame,p[0.077984, 0.140117, -0.000125, -0.013708, 3.141563, -0.000000]),accel_mss,speed_ms,0,0) # end trace
      speed_ms    = 0.007
      movel(pose_trans(ref_frame,p[0.090436, 0.140105, -0.000125, -0.013708, 3.141563, 0.000000]),accel_mss,speed_ms,0,0.001)
      movel(pose_trans(ref_frame,p[0.102888, 0.140092, -0.000125, -0.013708, 3.141563, 0.000000]),accel_mss,speed_ms,0,0.001)
      movel(pose_trans(ref_frame,p[0.113377, 0.140079, -0.000125, -0.013708, 3.141563, -0.000000]),accel_mss,speed_ms,0,0.001)
      movel(pose_trans(ref_frame,p[0.123866, 0.140064, -0.000125, -0.013708, 3.141563, -0.000000]),accel_mss,speed_ms,0,0.001)
      movel(pose_trans(ref_frame,p[0.142925, 0.140034, -0.000125, -0.013708, 3.141563, 0.000000]),accel_mss,speed_ms,0,0.001)
      movel(pose_trans(ref_frame,p[0.142963, 0.140030, -0.000125, -0.013708, 3.141563, -0.000000]),accel_mss,speed_ms,0,0.001)
      movel(pose_trans(ref_frame,p[0.142998, 0.140017, -0.000125, -0.013708, 3.141563, 0.000000]),accel_mss,speed_ms,0,0.001)
      movel(pose_trans(ref_frame,p[0.143094, 0.139929, -0.000125, -0.013708, 3.141563, 0.000000]),accel_mss,speed_ms,0,0.001)
      movel(pose_trans(ref_frame,p[0.143130, 0.139803, -0.000125, -0.013708, 3.141563, 0.000000]),accel_mss,speed_ms,0,0.001)
      movel(pose_trans(ref_frame,p[0.143174, 0.075002, -0.000125, -0.013708, 3.141563, 0.000000]),accel_mss,speed_ms,0,0.001)
      movel(pose_trans(ref_frame,p[0.143218, 0.010239, -0.000125, -0.013708, 3.141563, 0.000000]),accel_mss,speed_ms,0,0.001)
      movel(pose_trans(ref_frame,p[0.143185, 0.010068, -0.000125, -0.013708, 3.141563, -0.000000]),accel_mss,speed_ms,0,0.001)
      movel(pose_trans(ref_frame,p[0.143088, 0.009923, -0.000125, -0.013708, 3.141563, -0.000000]),accel_mss,speed_ms,0,0.001)
      movel(pose_trans(ref_frame,p[0.143041, 0.009891, -0.000125, -0.013708, 3.141563, -0.000000]),accel_mss,speed_ms,0,0.001)
      movel(pose_trans(ref_frame,p[0.142987, 0.009881, -0.000125, -0.013708, 3.141563, -0.000000]),accel_mss,speed_ms,0,0.001)
      movel(pose_trans(ref_frame,p[0.134476, 0.009866, -0.000125, -0.013708, 3.141563, 0.000000]),accel_mss,speed_ms,0,0.001)
      movel(pose_trans(ref_frame,p[0.129772, 0.009860, -0.000125, -0.013708, 3.141563, 0.000000]),accel_mss,speed_ms,0,0.001)
      movel(pose_trans(ref_frame,p[0.125068, 0.009860, -0.000125, -0.013708, 3.141563, 0.000000]),accel_mss,speed_ms,0,0.001)
      movel(pose_trans(ref_frame,p[0.119491, 0.009864, -0.000125, -0.013708, 3.141563, -0.000000]),accel_mss,speed_ms,0,0.001)
      movel(pose_trans(ref_frame,p[0.113913, 0.009873, -0.000125, -0.013708, 3.141563, -0.000000]),accel_mss,speed_ms,0,0.001)
      movel(pose_trans(ref_frame,p[0.107069, 0.009884, -0.000125, -0.013708, 3.141563, 0.000000]),accel_mss,speed_ms,0,0.001)
      movel(pose_trans(ref_frame,p[0.100224, 0.009893, -0.000125, -0.013708, 3.141563, -0.000000]),accel_mss,speed_ms,0,0.001)
      movel(pose_trans(ref_frame,p[0.091542, 0.009902, -0.000125, -0.013708, 3.141563, -0.000000]),accel_mss,speed_ms,0,0.001)
      movel(pose_trans(ref_frame,p[0.082859, 0.009909, -0.000125, -0.013708, 3.141563, 0.000000]),accel_mss,speed_ms,0,0.001)
      movel(pose_trans(ref_frame,p[0.073857, 0.009915, -0.000125, -0.013708, 3.141563, -0.000000]),accel_mss,speed_ms,0,0.001)
      movel(pose_trans(ref_frame,p[0.064855, 0.009920, -0.000125, -0.013708, 3.141563, -0.000000]),accel_mss,speed_ms,0,0.001)
      movel(pose_trans(ref_frame,p[0.056938, 0.009923, -0.000125, -0.013708, 3.141563, 0.000000]),accel_mss,speed_ms,0,0.001)
      movel(pose_trans(ref_frame,p[0.049021, 0.009923, -0.000125, -0.013708, 3.141563, -0.000000]),accel_mss,speed_ms,0,0.001)
      movel(pose_trans(ref_frame,p[0.042150, 0.009925, -0.000125, -0.013708, 3.141563, -0.000000]),accel_mss,speed_ms,0,0.001)
      movel(pose_trans(ref_frame,p[0.035278, 0.009930, -0.000125, -0.013708, 3.141563, -0.000000]),accel_mss,speed_ms,0,0.001)
      movel(pose_trans(ref_frame,p[0.029485, 0.009938, -0.000125, -0.013708, 3.141563, 0.000000]),accel_mss,speed_ms,0,0.001)
      movel(pose_trans(ref_frame,p[0.023692, 0.009951, -0.000125, -0.013708, 3.141563, 0.000000]),accel_mss,speed_ms,0,0.001)
      movel(pose_trans(ref_frame,p[0.013198, 0.009980, -0.000125, -0.013708, 3.141563, 0.000000]),accel_mss,speed_ms,0,0.001)
      movel(pose_trans(ref_frame,p[0.013144, 0.009991, -0.000125, -0.013708, 3.141563, 0.000000]),accel_mss,speed_ms,0,0.001)
      movel(pose_trans(ref_frame,p[0.013097, 0.010021, -0.000125, -0.013708, 3.141563, -0.000000]),accel_mss,speed_ms,0,0.001)
      movel(pose_trans(ref_frame,p[0.013051, 0.010089, -0.000125, -0.013708, 3.141563, 0.000000]),accel_mss,speed_ms,0,0.001)
      movel(pose_trans(ref_frame,p[0.013034, 0.010169, -0.000125, -0.013708, 3.141563, 0.000000]),accel_mss,speed_ms,0,0.001)
      movel(pose_trans(ref_frame,p[0.012995, 0.038219, -0.000125, -0.013708, 3.141563, 0.000000]),accel_mss,speed_ms,0,0.001)
      movel(pose_trans(ref_frame,p[0.012973, 0.056564, -0.000125, -0.013708, 3.141563, 0.000000]),accel_mss,speed_ms,0,0.001)
      movel(pose_trans(ref_frame,p[0.012958, 0.074909, -0.000125, -0.013708, 3.141563, 0.000000]),accel_mss,speed_ms,0,0.001)
      movel(pose_trans(ref_frame,p[0.012940, 0.104584, -0.000125, -0.013708, 3.141563, 0.000000]),accel_mss,speed_ms,0,0.001)
      movel(pose_trans(ref_frame,p[0.012925, 0.134259, -0.000125, -0.013708, 3.141563, 0.000000]),accel_mss,speed_ms,0,0.001)
      movel(pose_trans(ref_frame,p[0.012925, 0.135370, -0.000125, -0.013708, 3.141563, 0.000000]),accel_mss,speed_ms,0,0.001)
      movel(pose_trans(ref_frame,p[0.012928, 0.136481, -0.000125, -0.013708, 3.141563, -0.000000]),accel_mss,speed_ms,0,0.001)
      movel(pose_trans(ref_frame,p[0.012934, 0.137422, -0.000125, -0.013708, 3.141563, 0.000000]),accel_mss,speed_ms,0,0.001)
      movel(pose_trans(ref_frame,p[0.012942, 0.138363, -0.000125, -0.013708, 3.141563, 0.000000]),accel_mss,speed_ms,0,0.001)
      movel(pose_trans(ref_frame,p[0.012951, 0.139203, -0.000125, -0.013708, 3.141563, -0.000000]),accel_mss,speed_ms,0,0.001)
      movel(pose_trans(ref_frame,p[0.012961, 0.140044, -0.000125, -0.013708, 3.141563, 0.000000]),accel_mss,speed_ms,0,0.001)
      movel(pose_trans(ref_frame,p[0.012968, 0.140078, -0.000125, -0.013708, 3.141563, -0.000000]),accel_mss,speed_ms,0,0.001)
      movel(pose_trans(ref_frame,p[0.012988, 0.140108, -0.000125, -0.013708, 3.141563, 0.000000]),accel_mss,speed_ms,0,0.001)
      movel(pose_trans(ref_frame,p[0.013018, 0.140128, -0.000125, -0.013708, 3.141563, 0.000000]),accel_mss,speed_ms,0,0.001)
      movel(pose_trans(ref_frame,p[0.013054, 0.140135, -0.000125, -0.013708, 3.141563, 0.000000]),accel_mss,speed_ms,0,0.001)
      movel(pose_trans(ref_frame,p[0.032108, 0.140138, -0.000125, -0.013708, 3.141563, 0.000000]),accel_mss,speed_ms,0,0.001)
      movel(pose_trans(ref_frame,p[0.042595, 0.140137, -0.000125, -0.013708, 3.141563, 0.000000]),accel_mss,speed_ms,0,0.001)
      movel(pose_trans(ref_frame,p[0.053082, 0.140134, -0.000125, -0.013708, 3.141563, 0.000000]),accel_mss,speed_ms,0,0.001)
      movel(pose_trans(ref_frame,p[0.065533, 0.140126, -0.000125, -0.013708, 3.141563, -0.000000]),accel_mss,speed_ms,0,0.001)
      movel(pose_trans(ref_frame,p[0.077984, 0.140117, -0.000125, -0.013708, 3.141563, -0.000000]),accel_mss,speed_ms,0,0) # end trace
      speed_ms    = 1.000
      movel(pose_trans(ref_frame,p[0.077984, 0.140117, 0.005000, -0.013708, 3.141563, 0.000000]),accel_mss,speed_ms,0,0.001)
      movel(pose_trans(ref_frame,p[0.084325, 0.132557, 0.005000, -0.013708, 3.141563, 0.000000]),accel_mss,speed_ms,0,0) # end trace
      speed_ms    = 0.002
      movel(pose_trans(ref_frame,p[0.084325, 0.132557, -0.000125, -0.013708, 3.141563, 0.000000]),accel_mss,speed_ms,0,0) # end trace
      speed_ms    = 0.007
      movel(pose_trans(ref_frame,p[0.084424, 0.132582, -0.000125, -0.013708, 3.141563, -0.000000]),accel_mss,speed_ms,0,0.001)
      movel(pose_trans(ref_frame,p[0.084525, 0.132596, -0.000125, -0.013708, 3.141563, -0.000000]),accel_mss,speed_ms,0,0.001)
      movel(pose_trans(ref_frame,p[0.084623, 0.132598, -0.000125, -0.013708, 3.141563, 0.000000]),accel_mss,speed_ms,0,0.001)
      movel(pose_trans(ref_frame,p[0.084721, 0.132588, -0.000125, -0.013708, 3.141563, 0.000000]),accel_mss,speed_ms,0,0.001)
      movel(pose_trans(ref_frame,p[0.084826, 0.132564, -0.000125, -0.013708, 3.141563, 0.000000]),accel_mss,speed_ms,0,0.001)
      movel(pose_trans(ref_frame,p[0.084928, 0.132528, -0.000125, -0.013708, 3.141563, 0.000000]),accel_mss,speed_ms,0,0.001)
      movel(pose_trans(ref_frame,p[0.085047, 0.132474, -0.000125, -0.013708, 3.141563, -0.000000]),accel_mss,speed_ms,0,0.001)
      movel(pose_trans(ref_frame,p[0.085162, 0.132413, -0.000125, -0.013708, 3.141563, 0.000000]),accel_mss,speed_ms,0,0.001)
      movel(pose_trans(ref_frame,p[0.085840, 0.132038, -0.000125, -0.013708, 3.141563, 0.000000]),accel_mss,speed_ms,0,0.001)
      movel(pose_trans(ref_frame,p[0.086528, 0.131682, -0.000125, -0.013708, 3.141563, -0.000000]),accel_mss,speed_ms,0,0.001)
      movel(pose_trans(ref_frame,p[0.087108, 0.131411, -0.000125, -0.013708, 3.141563, 0.000000]),accel_mss,speed_ms,0,0.001)
      movel(pose_trans(ref_frame,p[0.087700, 0.131168, -0.000125, -0.013708, 3.141563, -0.000000]),accel_mss,speed_ms,0,0.001)
      movel(pose_trans(ref_frame,p[0.088195, 0.130997, -0.000125, -0.013708, 3.141563, 0.000000]),accel_mss,speed_ms,0,0.001)
      movel(pose_trans(ref_frame,p[0.088700, 0.130855, -0.000125, -0.013708, 3.141563, 0.000000]),accel_mss,speed_ms,0,0.001)
      movel(pose_trans(ref_frame,p[0.089112, 0.130778, -0.000125, -0.013708, 3.141563, 0.000000]),accel_mss,speed_ms,0,0.001)
      movel(pose_trans(ref_frame,p[0.089531, 0.130750, -0.000125, -0.013708, 3.141563, -0.000000]),accel_mss,speed_ms,0,0.001)
      movel(pose_trans(ref_frame,p[0.089908, 0.130765, -0.000125, -0.013708, 3.141563, -0.000000]),accel_mss,speed_ms,0,0.001)
      movel(pose_trans(ref_frame,p[0.090282, 0.130819, -0.000125, -0.013708, 3.141563, 0.000000]),accel_mss,speed_ms,0,0.001)
      movel(pose_trans(ref_frame,p[0.090720, 0.130919, -0.000125, -0.013708, 3.141563, 0.000000]),accel_mss,speed_ms,0,0.001)
      movel(pose_trans(ref_frame,p[0.091151, 0.131045, -0.000125, -0.013708, 3.141563, -0.000000]),accel_mss,speed_ms,0,0.001)
      movel(pose_trans(ref_frame,p[0.091637, 0.131217, -0.000125, -0.013708, 3.141563, 0.000000]),accel_mss,speed_ms,0,0.001)
      movel(pose_trans(ref_frame,p[0.092112, 0.131415, -0.000125, -0.013708, 3.141563, -0.000000]),accel_mss,speed_ms,0,0.001)
      movel(pose_trans(ref_frame,p[0.092632, 0.131660, -0.000125, -0.013708, 3.141563, 0.000000]),accel_mss,speed_ms,0,0.001)
      movel(pose_trans(ref_frame,p[0.093141, 0.131925, -0.000125, -0.013708, 3.141563, 0.000000]),accel_mss,speed_ms,0,0.001)
      movel(pose_trans(ref_frame,p[0.093583, 0.132155, -0.000125, -0.013708, 3.141563, 0.000000]),accel_mss,speed_ms,0,0.001)
      movel(pose_trans(ref_frame,p[0.094033, 0.132367, -0.000125, -0.013708, 3.141563, 0.000000]),accel_mss,speed_ms,0,0.001)
      movel(pose_trans(ref_frame,p[0.094322, 0.132471, -0.000125, -0.013708, 3.141563, 0.000000]),accel_mss,speed_ms,0,0.001)
      movel(pose_trans(ref_frame,p[0.094623, 0.132531, -0.000125, -0.013708, 3.141563, -0.000000]),accel_mss,speed_ms,0,0.001)
      movel(pose_trans(ref_frame,p[0.094836, 0.132527, -0.000125, -0.013708, 3.141563, 0.000000]),accel_mss,speed_ms,0,0.001)
      movel(pose_trans(ref_frame,p[0.095041, 0.132465, -0.000125, -0.013708, 3.141563, 0.000000]),accel_mss,speed_ms,0,0.001)
      movel(pose_trans(ref_frame,p[0.095220, 0.132351, -0.000125, -0.013708, 3.141563, 0.000000]),accel_mss,speed_ms,0,0.001)
      movel(pose_trans(ref_frame,p[0.095361, 0.132192, -0.000125, -0.013708, 3.141563, -0.000000]),accel_mss,speed_ms,0,0.001)
      movel(pose_trans(ref_frame,p[0.095456, 0.132027, -0.000125, -0.013708, 3.141563, 0.000000]),accel_mss,speed_ms,0,0.001)
      movel(pose_trans(ref_frame,p[0.095526, 0.131851, -0.000125, -0.013708, 3.141563, -0.000000]),accel_mss,speed_ms,0,0.001)
      movel(pose_trans(ref_frame,p[0.095559, 0.131690, -0.000125, -0.013708, 3.141563, -0.000000]),accel_mss,speed_ms,0,0.001)
      movel(pose_trans(ref_frame,p[0.095557, 0.131526, -0.000125, -0.013708, 3.141563, 0.000000]),accel_mss,speed_ms,0,0.001)
      movel(pose_trans(ref_frame,p[0.095519, 0.131332, -0.000125, -0.013708, 3.141563, 0.000000]),accel_mss,speed_ms,0,0.001)
      movel(pose_trans(ref_frame,p[0.095451, 0.131147, -0.000125, -0.013708, 3.141563, -0.000000]),accel_mss,speed_ms,0,0.001)
      movel(pose_trans(ref_frame,p[0.095319, 0.130876, -0.000125, -0.013708, 3.141563, 0.000000]),accel_mss,speed_ms,0,0.001)
      movel(pose_trans(ref_frame,p[0.095174, 0.130613, -0.000125, -0.013708, 3.141563, -0.000000]),accel_mss,speed_ms,0,0.001)
      movel(pose_trans(ref_frame,p[0.094821, 0.129970, -0.000125, -0.013708, 3.141563, 0.000000]),accel_mss,speed_ms,0,0.001)
      movel(pose_trans(ref_frame,p[0.094497, 0.129313, -0.000125, -0.013708, 3.141563, 0.000000]),accel_mss,speed_ms,0,0.001)
      movel(pose_trans(ref_frame,p[0.094241, 0.128711, -0.000125, -0.013708, 3.141563, -0.000000]),accel_mss,speed_ms,0,0.001)
      movel(pose_trans(ref_frame,p[0.094022, 0.128094, -0.000125, -0.013708, 3.141563, 0.000000]),accel_mss,speed_ms,0,0.001)
      movel(pose_trans(ref_frame,p[0.093873, 0.127560, -0.000125, -0.013708, 3.141563, 0.000000]),accel_mss,speed_ms,0,0.001)
      movel(pose_trans(ref_frame,p[0.093762, 0.127015, -0.000125, -0.013708, 3.141563, -0.000000]),accel_mss,speed_ms,0,0.001)
      movel(pose_trans(ref_frame,p[0.093724, 0.126582, -0.000125, -0.013708, 3.141563, 0.000000]),accel_mss,speed_ms,0,0.001)
      movel(pose_trans(ref_frame,p[0.093749, 0.126148, -0.000125, -0.013708, 3.141563, 0.000000]),accel_mss,speed_ms,0,0.001)
      movel(pose_trans(ref_frame,p[0.093808, 0.125810, -0.000125, -0.013708, 3.141563, -0.000000]),accel_mss,speed_ms,0,0.001)
      movel(pose_trans(ref_frame,p[0.093890, 0.125477, -0.000125, -0.013708, 3.141563, 0.000000]),accel_mss,speed_ms,0,0.001)
      movel(pose_trans(ref_frame,p[0.094012, 0.125080, -0.000125, -0.013708, 3.141563, -0.000000]),accel_mss,speed_ms,0,0.001)
      movel(pose_trans(ref_frame,p[0.094151, 0.124689, -0.000125, -0.013708, 3.141563, -0.000000]),accel_mss,speed_ms,0,0.001)
      movel(pose_trans(ref_frame,p[0.094323, 0.124257, -0.000125, -0.013708, 3.141563, 0.000000]),accel_mss,speed_ms,0,0.001)
      movel(pose_trans(ref_frame,p[0.094512, 0.123832, -0.000125, -0.013708, 3.141563, -0.000000]),accel_mss,speed_ms,0,0.001)
      movel(pose_trans(ref_frame,p[0.094727, 0.123389, -0.000125, -0.013708, 3.141563, 0.000000]),accel_mss,speed_ms,0,0.001)
      movel(pose_trans(ref_frame,p[0.094955, 0.122953, -0.000125, -0.013708, 3.141563, 0.000000]),accel_mss,speed_ms,0,0.001)
      movel(pose_trans(ref_frame,p[0.095172, 0.122541, -0.000125, -0.013708, 3.141563, 0.000000]),accel_mss,speed_ms,0,0.001)
      movel(pose_trans(ref_frame,p[0.095374, 0.122121, -0.000125, -0.013708, 3.141563, 0.000000]),accel_mss,speed_ms,0,0.001)
      movel(pose_trans(ref_frame,p[0.095468, 0.121870, -0.000125, -0.013708, 3.141563, -0.000000]),accel_mss,speed_ms,0,0.001)
      movel(pose_trans(ref_frame,p[0.095523, 0.121608, -0.000125, -0.013708, 3.141563, 0.000000]),accel_mss,speed_ms,0,0.001)
      movel(pose_trans(ref_frame,p[0.095523, 0.121412, -0.000125, -0.013708, 3.141563, 0.000000]),accel_mss,speed_ms,0,0.001)
      movel(pose_trans(ref_frame,p[0.095471, 0.121222, -0.000125, -0.013708, 3.141563, -0.000000]),accel_mss,speed_ms,0,0.001)
      movel(pose_trans(ref_frame,p[0.095368, 0.121031, -0.000125, -0.013708, 3.141563, 0.000000]),accel_mss,speed_ms,0,0.001)
      movel(pose_trans(ref_frame,p[0.095230, 0.120863, -0.000125, -0.013708, 3.141563, -0.000000]),accel_mss,speed_ms,0,0.001)
      movel(pose_trans(ref_frame,p[0.095075, 0.120737, -0.000125, -0.013708, 3.141563, 0.000000]),accel_mss,speed_ms,0,0.001)
      movel(pose_trans(ref_frame,p[0.094898, 0.120647, -0.000125, -0.013708, 3.141563, 0.000000]),accel_mss,speed_ms,0,0.001)
      movel(pose_trans(ref_frame,p[0.094719, 0.120603, -0.000125, -0.013708, 3.141563, 0.000000]),accel_mss,speed_ms,0,0.001)
      movel(pose_trans(ref_frame,p[0.094535, 0.120608, -0.000125, -0.013708, 3.141563, 0.000000]),accel_mss,speed_ms,0,0.001)
      movel(pose_trans(ref_frame,p[0.094284, 0.120667, -0.000125, -0.013708, 3.141563, 0.000000]),accel_mss,speed_ms,0,0.001)
      movel(pose_trans(ref_frame,p[0.094045, 0.120761, -0.000125, -0.013708, 3.141563, 0.000000]),accel_mss,speed_ms,0,0.001)
      movel(pose_trans(ref_frame,p[0.093642, 0.120962, -0.000125, -0.013708, 3.141563, 0.000000]),accel_mss,speed_ms,0,0.001)
      movel(pose_trans(ref_frame,p[0.093245, 0.121176, -0.000125, -0.013708, 3.141563, -0.000000]),accel_mss,speed_ms,0,0.001)
      movel(pose_trans(ref_frame,p[0.092798, 0.121419, -0.000125, -0.013708, 3.141563, -0.000000]),accel_mss,speed_ms,0,0.001)
      movel(pose_trans(ref_frame,p[0.092348, 0.121655, -0.000125, -0.013708, 3.141563, 0.000000]),accel_mss,speed_ms,0,0.001)
      movel(pose_trans(ref_frame,p[0.092001, 0.121823, -0.000125, -0.013708, 3.141563, 0.000000]),accel_mss,speed_ms,0,0.001)
      movel(pose_trans(ref_frame,p[0.091649, 0.121977, -0.000125, -0.013708, 3.141563, -0.000000]),accel_mss,speed_ms,0,0.001)
      movel(pose_trans(ref_frame,p[0.091343, 0.122094, -0.000125, -0.013708, 3.141563, -0.000000]),accel_mss,speed_ms,0,0.001)
      movel(pose_trans(ref_frame,p[0.091032, 0.122195, -0.000125, -0.013708, 3.141563, 0.000000]),accel_mss,speed_ms,0,0.001)
      movel(pose_trans(ref_frame,p[0.090719, 0.122279, -0.000125, -0.013708, 3.141563, 0.000000]),accel_mss,speed_ms,0,0.001)
      movel(pose_trans(ref_frame,p[0.090403, 0.122347, -0.000125, -0.013708, 3.141563, 0.000000]),accel_mss,speed_ms,0,0.001)
      movel(pose_trans(ref_frame,p[0.089899, 0.122408, -0.000125, -0.013708, 3.141563, 0.000000]),accel_mss,speed_ms,0,0.001)
      movel(pose_trans(ref_frame,p[0.089391, 0.122405, -0.000125, -0.013708, 3.141563, 0.000000]),accel_mss,speed_ms,0,0.001)
      movel(pose_trans(ref_frame,p[0.088835, 0.122340, -0.000125, -0.013708, 3.141563, 0.000000]),accel_mss,speed_ms,0,0.001)
      movel(pose_trans(ref_frame,p[0.088288, 0.122223, -0.000125, -0.013708, 3.141563, -0.000000]),accel_mss,speed_ms,0,0.001)
      movel(pose_trans(ref_frame,p[0.087677, 0.122035, -0.000125, -0.013708, 3.141563, 0.000000]),accel_mss,speed_ms,0,0.001)
      movel(pose_trans(ref_frame,p[0.087082, 0.121797, -0.000125, -0.013708, 3.141563, -0.000000]),accel_mss,speed_ms,0,0.001)
      movel(pose_trans(ref_frame,p[0.086412, 0.121477, -0.000125, -0.013708, 3.141563, 0.000000]),accel_mss,speed_ms,0,0.001)
      movel(pose_trans(ref_frame,p[0.085760, 0.121121, -0.000125, -0.013708, 3.141563, 0.000000]),accel_mss,speed_ms,0,0.001)
      movel(pose_trans(ref_frame,p[0.085441, 0.120949, -0.000125, -0.013708, 3.141563, 0.000000]),accel_mss,speed_ms,0,0.001)
      movel(pose_trans(ref_frame,p[0.085112, 0.120795, -0.000125, -0.013708, 3.141563, -0.000000]),accel_mss,speed_ms,0,0.001)
      movel(pose_trans(ref_frame,p[0.084863, 0.120709, -0.000125, -0.013708, 3.141563, 0.000000]),accel_mss,speed_ms,0,0.001)
      movel(pose_trans(ref_frame,p[0.084604, 0.120661, -0.000125, -0.013708, 3.141563, -0.000000]),accel_mss,speed_ms,0,0.001)
      movel(pose_trans(ref_frame,p[0.084398, 0.120660, -0.000125, -0.013708, 3.141563, -0.000000]),accel_mss,speed_ms,0,0.001)
      movel(pose_trans(ref_frame,p[0.084197, 0.120703, -0.000125, -0.013708, 3.141563, 0.000000]),accel_mss,speed_ms,0,0.001)
      movel(pose_trans(ref_frame,p[0.084016, 0.120787, -0.000125, -0.013708, 3.141563, -0.000000]),accel_mss,speed_ms,0,0.001)
      movel(pose_trans(ref_frame,p[0.083859, 0.120910, -0.000125, -0.013708, 3.141563, 0.000000]),accel_mss,speed_ms,0,0.001)
      movel(pose_trans(ref_frame,p[0.083733, 0.121067, -0.000125, -0.013708, 3.141563, -0.000000]),accel_mss,speed_ms,0,0.001)
      movel(pose_trans(ref_frame,p[0.083645, 0.121248, -0.000125, -0.013708, 3.141563, -0.000000]),accel_mss,speed_ms,0,0.001)
      movel(pose_trans(ref_frame,p[0.083604, 0.121436, -0.000125, -0.013708, 3.141563, 0.000000]),accel_mss,speed_ms,0,0.001)
      movel(pose_trans(ref_frame,p[0.083611, 0.121628, -0.000125, -0.013708, 3.141563, 0.000000]),accel_mss,speed_ms,0,0.001)
      movel(pose_trans(ref_frame,p[0.083672, 0.121890, -0.000125, -0.013708, 3.141563, -0.000000]),accel_mss,speed_ms,0,0.001)
      movel(pose_trans(ref_frame,p[0.083770, 0.122141, -0.000125, -0.013708, 3.141563, -0.000000]),accel_mss,speed_ms,0,0.001)
      movel(pose_trans(ref_frame,p[0.083972, 0.122549, -0.000125, -0.013708, 3.141563, 0.000000]),accel_mss,speed_ms,0,0.001)
      movel(pose_trans(ref_frame,p[0.084187, 0.122950, -0.000125, -0.013708, 3.141563, 0.000000]),accel_mss,speed_ms,0,0.001)
      movel(pose_trans(ref_frame,p[0.084686, 0.123932, -0.000125, -0.013708, 3.141563, 0.000000]),accel_mss,speed_ms,0,0.001)
      movel(pose_trans(ref_frame,p[0.085109, 0.124950, -0.000125, -0.013708, 3.141563, 0.000000]),accel_mss,speed_ms,0,0.001)
      movel(pose_trans(ref_frame,p[0.085329, 0.125752, -0.000125, -0.013708, 3.141563, -0.000000]),accel_mss,speed_ms,0,0.001)
      movel(pose_trans(ref_frame,p[0.085407, 0.126579, -0.000125, -0.013708, 3.141563, 0.000000]),accel_mss,speed_ms,0,0.001)
      movel(pose_trans(ref_frame,p[0.085341, 0.127402, -0.000125, -0.013708, 3.141563, -0.000000]),accel_mss,speed_ms,0,0.001)
      movel(pose_trans(ref_frame,p[0.085131, 0.128200, -0.000125, -0.013708, 3.141563, 0.000000]),accel_mss,speed_ms,0,0.001)
      movel(pose_trans(ref_frame,p[0.084724, 0.129203, -0.000125, -0.013708, 3.141563, 0.000000]),accel_mss,speed_ms,0,0.001)
      movel(pose_trans(ref_frame,p[0.084239, 0.130169, -0.000125, -0.013708, 3.141563, 0.000000]),accel_mss,speed_ms,0,0.001)
      movel(pose_trans(ref_frame,p[0.084015, 0.130580, -0.000125, -0.013708, 3.141563, -0.000000]),accel_mss,speed_ms,0,0.001)
      movel(pose_trans(ref_frame,p[0.083795, 0.130993, -0.000125, -0.013708, 3.141563, 0.000000]),accel_mss,speed_ms,0,0.001)
      movel(pose_trans(ref_frame,p[0.083699, 0.131193, -0.000125, -0.013708, 3.141563, 0.000000]),accel_mss,speed_ms,0,0.001)
      movel(pose_trans(ref_frame,p[0.083618, 0.131401, -0.000125, -0.013708, 3.141563, 0.000000]),accel_mss,speed_ms,0,0.001)
      movel(pose_trans(ref_frame,p[0.083583, 0.131539, -0.000125, -0.013708, 3.141563, 0.000000]),accel_mss,speed_ms,0,0.001)
      movel(pose_trans(ref_frame,p[0.083572, 0.131681, -0.000125, -0.013708, 3.141563, 0.000000]),accel_mss,speed_ms,0,0.001)
      movel(pose_trans(ref_frame,p[0.083586, 0.131814, -0.000125, -0.013708, 3.141563, -0.000000]),accel_mss,speed_ms,0,0.001)
      movel(pose_trans(ref_frame,p[0.083626, 0.131943, -0.000125, -0.013708, 3.141563, 0.000000]),accel_mss,speed_ms,0,0.001)
      movel(pose_trans(ref_frame,p[0.083683, 0.132066, -0.000125, -0.013708, 3.141563, 0.000000]),accel_mss,speed_ms,0,0.001)
      movel(pose_trans(ref_frame,p[0.083749, 0.132186, -0.000125, -0.013708, 3.141563, -0.000000]),accel_mss,speed_ms,0,0.001)
      movel(pose_trans(ref_frame,p[0.083807, 0.132269, -0.000125, -0.013708, 3.141563, 0.000000]),accel_mss,speed_ms,0,0.001)
      movel(pose_trans(ref_frame,p[0.083877, 0.132341, -0.000125, -0.013708, 3.141563, 0.000000]),accel_mss,speed_ms,0,0.001)
      movel(pose_trans(ref_frame,p[0.083960, 0.132403, -0.000125, -0.013708, 3.141563, -0.000000]),accel_mss,speed_ms,0,0.001)
      movel(pose_trans(ref_frame,p[0.084051, 0.132452, -0.000125, -0.013708, 3.141563, 0.000000]),accel_mss,speed_ms,0,0.001)
      movel(pose_trans(ref_frame,p[0.084186, 0.132508, -0.000125, -0.013708, 3.141563, -0.000000]),accel_mss,speed_ms,0,0.001)
      movel(pose_trans(ref_frame,p[0.084325, 0.132557, -0.000125, -0.013708, 3.141563, 0.000000]),accel_mss,speed_ms,0,0) # end trace
      speed_ms    = 1.000
      movel(pose_trans(ref_frame,p[0.084325, 0.132557, 0.005000, -0.013708, 3.141563, 0.000000]),accel_mss,speed_ms,0,0.001)
      movel(pose_trans(ref_frame,p[0.113210, 0.120470, 0.005000, -0.013708, 3.141563, -0.000000]),accel_mss,speed_ms,0,0) # end trace
      speed_ms    = 0.002
      movel(pose_trans(ref_frame,p[0.113210, 0.120470, -0.000125, -0.013708, 3.141563, -0.000000]),accel_mss,speed_ms,0,0) # end trace
      speed_ms    = 0.007
      movel(pose_trans(ref_frame,p[0.113719, 0.120766, -0.000125, -0.013708, 3.141563, 0.000000]),accel_mss,speed_ms,0,0.001)
      movel(pose_trans(ref_frame,p[0.114250, 0.121019, -0.000125, -0.013708, 3.141563, -0.000000]),accel_mss,speed_ms,0,0.001)
      movel(pose_trans(ref_frame,p[0.114778, 0.121216, -0.000125, -0.013708, 3.141563, -0.000000]),accel_mss,speed_ms,0,0.001)
      movel(pose_trans(ref_frame,p[0.115322, 0.121361, -0.000125, -0.013708, 3.141563, -0.000000]),accel_mss,speed_ms,0,0.001)
      movel(pose_trans(ref_frame,p[0.115827, 0.121444, -0.000125, -0.013708, 3.141563, 0.000000]),accel_mss,speed_ms,0,0.001)
      movel(pose_trans(ref_frame,p[0.116338, 0.121473, -0.000125, -0.013708, 3.141563, -0.000000]),accel_mss,speed_ms,0,0.001)
      movel(pose_trans(ref_frame,p[0.116780, 0.121440, -0.000125, -0.013708, 3.141563, 0.000000]),accel_mss,speed_ms,0,0.001)
      movel(pose_trans(ref_frame,p[0.117211, 0.121338, -0.000125, -0.013708, 3.141563, 0.000000]),accel_mss,speed_ms,0,0.001)
      movel(pose_trans(ref_frame,p[0.117501, 0.121226, -0.000125, -0.013708, 3.141563, -0.000000]),accel_mss,speed_ms,0,0.001)
      movel(pose_trans(ref_frame,p[0.117778, 0.121084, -0.000125, -0.013708, 3.141563, 0.000000]),accel_mss,speed_ms,0,0.001)
      movel(pose_trans(ref_frame,p[0.118088, 0.120890, -0.000125, -0.013708, 3.141563, -0.000000]),accel_mss,speed_ms,0,0.001)
      movel(pose_trans(ref_frame,p[0.118384, 0.120676, -0.000125, -0.013708, 3.141563, -0.000000]),accel_mss,speed_ms,0,0.001)
      movel(pose_trans(ref_frame,p[0.118673, 0.120437, -0.000125, -0.013708, 3.141563, 0.000000]),accel_mss,speed_ms,0,0.001)
      movel(pose_trans(ref_frame,p[0.118945, 0.120180, -0.000125, -0.013708, 3.141563, 0.000000]),accel_mss,speed_ms,0,0.001)
      movel(pose_trans(ref_frame,p[0.119171, 0.119931, -0.000125, -0.013708, 3.141563, 0.000000]),accel_mss,speed_ms,0,0.001)
      movel(pose_trans(ref_frame,p[0.119375, 0.119662, -0.000125, -0.013708, 3.141563, 0.000000]),accel_mss,speed_ms,0,0.001)
      movel(pose_trans(ref_frame,p[0.119636, 0.119239, -0.000125, -0.013708, 3.141563, -0.000000]),accel_mss,speed_ms,0,0.001)
      movel(pose_trans(ref_frame,p[0.119852, 0.118791, -0.000125, -0.013708, 3.141563, 0.000000]),accel_mss,speed_ms,0,0.001)
      movel(pose_trans(ref_frame,p[0.120026, 0.118314, -0.000125, -0.013708, 3.141563, 0.000000]),accel_mss,speed_ms,0,0.001)
      movel(pose_trans(ref_frame,p[0.120152, 0.117823, -0.000125, -0.013708, 3.141563, 0.000000]),accel_mss,speed_ms,0,0.001)
      movel(pose_trans(ref_frame,p[0.120259, 0.117196, -0.000125, -0.013708, 3.141563, 0.000000]),accel_mss,speed_ms,0,0.001)
      movel(pose_trans(ref_frame,p[0.120322, 0.116563, -0.000125, -0.013708, 3.141563, -0.000000]),accel_mss,speed_ms,0,0.001)
      movel(pose_trans(ref_frame,p[0.120370, 0.115646, -0.000125, -0.013708, 3.141563, 0.000000]),accel_mss,speed_ms,0,0.001)
      movel(pose_trans(ref_frame,p[0.120395, 0.114729, -0.000125, -0.013708, 3.141563, 0.000000]),accel_mss,speed_ms,0,0.001)
      movel(pose_trans(ref_frame,p[0.120405, 0.114223, -0.000125, -0.013708, 3.141563, 0.000000]),accel_mss,speed_ms,0,0.001)
      movel(pose_trans(ref_frame,p[0.120419, 0.113717, -0.000125, -0.013708, 3.141563, -0.000000]),accel_mss,speed_ms,0,0.001)
      movel(pose_trans(ref_frame,p[0.120437, 0.113239, -0.000125, -0.013708, 3.141563, 0.000000]),accel_mss,speed_ms,0,0.001)
      movel(pose_trans(ref_frame,p[0.120460, 0.112761, -0.000125, -0.013708, 3.141563, 0.000000]),accel_mss,speed_ms,0,0.001)
      movel(pose_trans(ref_frame,p[0.120482, 0.112357, -0.000125, -0.013708, 3.141563, -0.000000]),accel_mss,speed_ms,0,0.001)
      movel(pose_trans(ref_frame,p[0.120508, 0.111954, -0.000125, -0.013708, 3.141563, 0.000000]),accel_mss,speed_ms,0,0.001)
      movel(pose_trans(ref_frame,p[0.120528, 0.111760, -0.000125, -0.013708, 3.141563, -0.000000]),accel_mss,speed_ms,0,0.001)
      movel(pose_trans(ref_frame,p[0.120559, 0.111566, -0.000125, -0.013708, 3.141563, 0.000000]),accel_mss,speed_ms,0,0.001)
      movel(pose_trans(ref_frame,p[0.120613, 0.111321, -0.000125, -0.013708, 3.141563, 0.000000]),accel_mss,speed_ms,0,0.001)
      movel(pose_trans(ref_frame,p[0.120679, 0.111078, -0.000125, -0.013708, 3.141563, -0.000000]),accel_mss,speed_ms,0,0.001)
      movel(pose_trans(ref_frame,p[0.120766, 0.110804, -0.000125, -0.013708, 3.141563, 0.000000]),accel_mss,speed_ms,0,0.001)
      movel(pose_trans(ref_frame,p[0.120863, 0.110533, -0.000125, -0.013708, 3.141563, 0.000000]),accel_mss,speed_ms,0,0.001)
      movel(pose_trans(ref_frame,p[0.120959, 0.110287, -0.000125, -0.013708, 3.141563, -0.000000]),accel_mss,speed_ms,0,0.001)
      movel(pose_trans(ref_frame,p[0.121061, 0.110044, -0.000125, -0.013708, 3.141563, 0.000000]),accel_mss,speed_ms,0,0.001)
      movel(pose_trans(ref_frame,p[0.121126, 0.109928, -0.000125, -0.013708, 3.141563, 0.000000]),accel_mss,speed_ms,0,0.001)
      movel(pose_trans(ref_frame,p[0.121210, 0.109826, -0.000125, -0.013708, 3.141563, 0.000000]),accel_mss,speed_ms,0,0.001)
      movel(pose_trans(ref_frame,p[0.121274, 0.109785, -0.000125, -0.013708, 3.141563, -0.000000]),accel_mss,speed_ms,0,0.001)
      movel(pose_trans(ref_frame,p[0.121350, 0.109772, -0.000125, -0.013708, 3.141563, 0.000000]),accel_mss,speed_ms,0,0.001)
      movel(pose_trans(ref_frame,p[0.121424, 0.109792, -0.000125, -0.013708, 3.141563, 0.000000]),accel_mss,speed_ms,0,0.001)
      movel(pose_trans(ref_frame,p[0.121484, 0.109840, -0.000125, -0.013708, 3.141563, 0.000000]),accel_mss,speed_ms,0,0.001)
      movel(pose_trans(ref_frame,p[0.121845, 0.110297, -0.000125, -0.013708, 3.141563, -0.000000]),accel_mss,speed_ms,0,0.001)
      movel(pose_trans(ref_frame,p[0.122191, 0.110766, -0.000125, -0.013708, 3.141563, -0.000000]),accel_mss,speed_ms,0,0.001)
      movel(pose_trans(ref_frame,p[0.122535, 0.111273, -0.000125, -0.013708, 3.141563, 0.000000]),accel_mss,speed_ms,0,0.001)
      movel(pose_trans(ref_frame,p[0.122854, 0.111796, -0.000125, -0.013708, 3.141563, -0.000000]),accel_mss,speed_ms,0,0.001)
      movel(pose_trans(ref_frame,p[0.123057, 0.112201, -0.000125, -0.013708, 3.141563, 0.000000]),accel_mss,speed_ms,0,0.001)
      movel(pose_trans(ref_frame,p[0.123210, 0.112627, -0.000125, -0.013708, 3.141563, 0.000000]),accel_mss,speed_ms,0,0.001)
      movel(pose_trans(ref_frame,p[0.123290, 0.112955, -0.000125, -0.013708, 3.141563, 0.000000]),accel_mss,speed_ms,0,0.001)
      movel(pose_trans(ref_frame,p[0.123340, 0.113289, -0.000125, -0.013708, 3.141563, 0.000000]),accel_mss,speed_ms,0,0.001)
      movel(pose_trans(ref_frame,p[0.123361, 0.113637, -0.000125, -0.013708, 3.141563, 0.000000]),accel_mss,speed_ms,0,0.001)
      movel(pose_trans(ref_frame,p[0.123352, 0.113985, -0.000125, -0.013708, 3.141563, 0.000000]),accel_mss,speed_ms,0,0.001)
      movel(pose_trans(ref_frame,p[0.123315, 0.114327, -0.000125, -0.013708, 3.141563, -0.000000]),accel_mss,speed_ms,0,0.001)
      movel(pose_trans(ref_frame,p[0.123248, 0.114665, -0.000125, -0.013708, 3.141563, 0.000000]),accel_mss,speed_ms,0,0.001)
      movel(pose_trans(ref_frame,p[0.123156, 0.114976, -0.000125, -0.013708, 3.141563, 0.000000]),accel_mss,speed_ms,0,0.001)
      movel(pose_trans(ref_frame,p[0.123033, 0.115276, -0.000125, -0.013708, 3.141563, -0.000000]),accel_mss,speed_ms,0,0.001)
      movel(pose_trans(ref_frame,p[0.122957, 0.115444, -0.000125, -0.013708, 3.141563, 0.000000]),accel_mss,speed_ms,0,0.001)
      movel(pose_trans(ref_frame,p[0.122886, 0.115613, -0.000125, -0.013708, 3.141563, -0.000000]),accel_mss,speed_ms,0,0.001)
      movel(pose_trans(ref_frame,p[0.122854, 0.115711, -0.000125, -0.013708, 3.141563, -0.000000]),accel_mss,speed_ms,0,0.001)
      movel(pose_trans(ref_frame,p[0.122838, 0.115812, -0.000125, -0.013708, 3.141563, 0.000000]),accel_mss,speed_ms,0,0.001)
      movel(pose_trans(ref_frame,p[0.122840, 0.115887, -0.000125, -0.013708, 3.141563, -0.000000]),accel_mss,speed_ms,0,0.001)
      movel(pose_trans(ref_frame,p[0.122862, 0.115959, -0.000125, -0.013708, 3.141563, -0.000000]),accel_mss,speed_ms,0,0.001)
      movel(pose_trans(ref_frame,p[0.122904, 0.116032, -0.000125, -0.013708, 3.141563, -0.000000]),accel_mss,speed_ms,0,0.001)
      movel(pose_trans(ref_frame,p[0.122958, 0.116097, -0.000125, -0.013708, 3.141563, 0.000000]),accel_mss,speed_ms,0,0.001)
      movel(pose_trans(ref_frame,p[0.123170, 0.116310, -0.000125, -0.013708, 3.141563, -0.000000]),accel_mss,speed_ms,0,0.001)
      movel(pose_trans(ref_frame,p[0.124581, 0.114946, -0.000125, -0.013708, 3.141563, -0.000000]),accel_mss,speed_ms,0,0.001)
      movel(pose_trans(ref_frame,p[0.124881, 0.114653, -0.000125, -0.013708, 3.141563, -0.000000]),accel_mss,speed_ms,0,0.001)
      movel(pose_trans(ref_frame,p[0.125177, 0.114358, -0.000125, -0.013708, 3.141563, 0.000000]),accel_mss,speed_ms,0,0.001)
      movel(pose_trans(ref_frame,p[0.125410, 0.114119, -0.000125, -0.013708, 3.141563, 0.000000]),accel_mss,speed_ms,0,0.001)
      movel(pose_trans(ref_frame,p[0.125637, 0.113875, -0.000125, -0.013708, 3.141563, 0.000000]),accel_mss,speed_ms,0,0.001)
      movel(pose_trans(ref_frame,p[0.125809, 0.113685, -0.000125, -0.013708, 3.141563, 0.000000]),accel_mss,speed_ms,0,0.001)
      movel(pose_trans(ref_frame,p[0.125977, 0.113492, -0.000125, -0.013708, 3.141563, 0.000000]),accel_mss,speed_ms,0,0.001)
      movel(pose_trans(ref_frame,p[0.126033, 0.113411, -0.000125, -0.013708, 3.141563, 0.000000]),accel_mss,speed_ms,0,0.001)
      movel(pose_trans(ref_frame,p[0.126071, 0.113321, -0.000125, -0.013708, 3.141563, 0.000000]),accel_mss,speed_ms,0,0.001)
      movel(pose_trans(ref_frame,p[0.126078, 0.113184, -0.000125, -0.013708, 3.141563, -0.000000]),accel_mss,speed_ms,0,0.001)
      movel(pose_trans(ref_frame,p[0.126022, 0.113060, -0.000125, -0.013708, 3.141563, 0.000000]),accel_mss,speed_ms,0,0.001)
      movel(pose_trans(ref_frame,p[0.125807, 0.112796, -0.000125, -0.013708, 3.141563, -0.000000]),accel_mss,speed_ms,0,0.001)
      movel(pose_trans(ref_frame,p[0.125581, 0.112542, -0.000125, -0.013708, 3.141563, -0.000000]),accel_mss,speed_ms,0,0.001)
      movel(pose_trans(ref_frame,p[0.125132, 0.112070, -0.000125, -0.013708, 3.141563, -0.000000]),accel_mss,speed_ms,0,0.001)
      movel(pose_trans(ref_frame,p[0.124674, 0.111606, -0.000125, -0.013708, 3.141563, 0.000000]),accel_mss,speed_ms,0,0.001)
      movel(pose_trans(ref_frame,p[0.123303, 0.110245, -0.000125, -0.013708, 3.141563, 0.000000]),accel_mss,speed_ms,0,0.001)
      movel(pose_trans(ref_frame,p[0.121931, 0.108886, -0.000125, -0.013708, 3.141563, -0.000000]),accel_mss,speed_ms,0,0.001)
      movel(pose_trans(ref_frame,p[0.117712, 0.104711, -0.000125, -0.013708, 3.141563, 0.000000]),accel_mss,speed_ms,0,0.001)
      movel(pose_trans(ref_frame,p[0.117216, 0.105153, -0.000125, -0.013708, 3.141563, -0.000000]),accel_mss,speed_ms,0,0.001)
      movel(pose_trans(ref_frame,p[0.116804, 0.105585, -0.000125, -0.013708, 3.141563, 0.000000]),accel_mss,speed_ms,0,0.001)
      movel(pose_trans(ref_frame,p[0.116471, 0.106081, -0.000125, -0.013708, 3.141563, 0.000000]),accel_mss,speed_ms,0,0.001)
      movel(pose_trans(ref_frame,p[0.116207, 0.106647, -0.000125, -0.013708, 3.141563, 0.000000]),accel_mss,speed_ms,0,0.001)
      movel(pose_trans(ref_frame,p[0.116029, 0.107247, -0.000125, -0.013708, 3.141563, 0.000000]),accel_mss,speed_ms,0,0.001)
      movel(pose_trans(ref_frame,p[0.115876, 0.108114, -0.000125, -0.013708, 3.141563, -0.000000]),accel_mss,speed_ms,0,0.001)
      movel(pose_trans(ref_frame,p[0.115797, 0.108992, -0.000125, -0.013708, 3.141563, 0.000000]),accel_mss,speed_ms,0,0.001)
      movel(pose_trans(ref_frame,p[0.115739, 0.110498, -0.000125, -0.013708, 3.141563, 0.000000]),accel_mss,speed_ms,0,0.001)
      movel(pose_trans(ref_frame,p[0.115709, 0.112004, -0.000125, -0.013708, 3.141563, 0.000000]),accel_mss,speed_ms,0,0.001)
      movel(pose_trans(ref_frame,p[0.115686, 0.113478, -0.000125, -0.013708, 3.141563, -0.000000]),accel_mss,speed_ms,0,0.001)
      movel(pose_trans(ref_frame,p[0.115647, 0.114951, -0.000125, -0.013708, 3.141563, -0.000000]),accel_mss,speed_ms,0,0.001)
      movel(pose_trans(ref_frame,p[0.115598, 0.115684, -0.000125, -0.013708, 3.141563, -0.000000]),accel_mss,speed_ms,0,0.001)
      movel(pose_trans(ref_frame,p[0.115497, 0.116412, -0.000125, -0.013708, 3.141563, -0.000000]),accel_mss,speed_ms,0,0.001)
      movel(pose_trans(ref_frame,p[0.115378, 0.116886, -0.000125, -0.013708, 3.141563, -0.000000]),accel_mss,speed_ms,0,0.001)
      movel(pose_trans(ref_frame,p[0.115191, 0.117338, -0.000125, -0.013708, 3.141563, -0.000000]),accel_mss,speed_ms,0,0.001)
      movel(pose_trans(ref_frame,p[0.114947, 0.117742, -0.000125, -0.013708, 3.141563, 0.000000]),accel_mss,speed_ms,0,0.001)
      movel(pose_trans(ref_frame,p[0.114640, 0.118102, -0.000125, -0.013708, 3.141563, 0.000000]),accel_mss,speed_ms,0,0.001)
      movel(pose_trans(ref_frame,p[0.114375, 0.118334, -0.000125, -0.013708, 3.141563, -0.000000]),accel_mss,speed_ms,0,0.001)
      movel(pose_trans(ref_frame,p[0.114080, 0.118527, -0.000125, -0.013708, 3.141563, 0.000000]),accel_mss,speed_ms,0,0.001)
      movel(pose_trans(ref_frame,p[0.113792, 0.118654, -0.000125, -0.013708, 3.141563, -0.000000]),accel_mss,speed_ms,0,0.001)
      movel(pose_trans(ref_frame,p[0.113485, 0.118725, -0.000125, -0.013708, 3.141563, 0.000000]),accel_mss,speed_ms,0,0.001)
      movel(pose_trans(ref_frame,p[0.113183, 0.118735, -0.000125, -0.013708, 3.141563, -0.000000]),accel_mss,speed_ms,0,0.001)
      movel(pose_trans(ref_frame,p[0.112885, 0.118684, -0.000125, -0.013708, 3.141563, 0.000000]),accel_mss,speed_ms,0,0.001)
      movel(pose_trans(ref_frame,p[0.112588, 0.118572, -0.000125, -0.013708, 3.141563, 0.000000]),accel_mss,speed_ms,0,0.001)
      movel(pose_trans(ref_frame,p[0.112314, 0.118411, -0.000125, -0.013708, 3.141563, 0.000000]),accel_mss,speed_ms,0,0.001)
      movel(pose_trans(ref_frame,p[0.112167, 0.118294, -0.000125, -0.013708, 3.141563, -0.000000]),accel_mss,speed_ms,0,0.001)
      movel(pose_trans(ref_frame,p[0.112034, 0.118161, -0.000125, -0.013708, 3.141563, 0.000000]),accel_mss,speed_ms,0,0.001)
      movel(pose_trans(ref_frame,p[0.111917, 0.118015, -0.000125, -0.013708, 3.141563, 0.000000]),accel_mss,speed_ms,0,0.001)
      movel(pose_trans(ref_frame,p[0.111818, 0.117856, -0.000125, -0.013708, 3.141563, -0.000000]),accel_mss,speed_ms,0,0.001)
      movel(pose_trans(ref_frame,p[0.111755, 0.117719, -0.000125, -0.013708, 3.141563, 0.000000]),accel_mss,speed_ms,0,0.001)
      movel(pose_trans(ref_frame,p[0.111710, 0.117575, -0.000125, -0.013708, 3.141563, 0.000000]),accel_mss,speed_ms,0,0.001)
      movel(pose_trans(ref_frame,p[0.111712, 0.117481, -0.000125, -0.013708, 3.141563, 0.000000]),accel_mss,speed_ms,0,0.001)
      movel(pose_trans(ref_frame,p[0.111760, 0.117401, -0.000125, -0.013708, 3.141563, 0.000000]),accel_mss,speed_ms,0,0.001)
      movel(pose_trans(ref_frame,p[0.111795, 0.117370, -0.000125, -0.013708, 3.141563, 0.000000]),accel_mss,speed_ms,0,0.001)
      movel(pose_trans(ref_frame,p[0.111834, 0.117346, -0.000125, -0.013708, 3.141563, 0.000000]),accel_mss,speed_ms,0,0.001)
      movel(pose_trans(ref_frame,p[0.111925, 0.117297, -0.000125, -0.013708, 3.141563, -0.000000]),accel_mss,speed_ms,0,0.001)
      movel(pose_trans(ref_frame,p[0.112018, 0.117250, -0.000125, -0.013708, 3.141563, 0.000000]),accel_mss,speed_ms,0,0.001)
      movel(pose_trans(ref_frame,p[0.112130, 0.117195, -0.000125, -0.013708, 3.141563, 0.000000]),accel_mss,speed_ms,0,0.001)
      movel(pose_trans(ref_frame,p[0.112242, 0.117143, -0.000125, -0.013708, 3.141563, 0.000000]),accel_mss,speed_ms,0,0.001)
      movel(pose_trans(ref_frame,p[0.112365, 0.117089, -0.000125, -0.013708, 3.141563, 0.000000]),accel_mss,speed_ms,0,0.001)
      movel(pose_trans(ref_frame,p[0.112488, 0.117037, -0.000125, -0.013708, 3.141563, 0.000000]),accel_mss,speed_ms,0,0.001)
      movel(pose_trans(ref_frame,p[0.112829, 0.116861, -0.000125, -0.013708, 3.141563, 0.000000]),accel_mss,speed_ms,0,0.001)
      movel(pose_trans(ref_frame,p[0.113136, 0.116631, -0.000125, -0.013708, 3.141563, 0.000000]),accel_mss,speed_ms,0,0.001)
      movel(pose_trans(ref_frame,p[0.113379, 0.116366, -0.000125, -0.013708, 3.141563, -0.000000]),accel_mss,speed_ms,0,0.001)
      movel(pose_trans(ref_frame,p[0.113563, 0.116057, -0.000125, -0.013708, 3.141563, -0.000000]),accel_mss,speed_ms,0,0.001)
      movel(pose_trans(ref_frame,p[0.113678, 0.115725, -0.000125, -0.013708, 3.141563, 0.000000]),accel_mss,speed_ms,0,0.001)
      movel(pose_trans(ref_frame,p[0.113721, 0.115377, -0.000125, -0.013708, 3.141563, -0.000000]),accel_mss,speed_ms,0,0.001)
      movel(pose_trans(ref_frame,p[0.113694, 0.115014, -0.000125, -0.013708, 3.141563, 0.000000]),accel_mss,speed_ms,0,0.001)
      movel(pose_trans(ref_frame,p[0.113598, 0.114663, -0.000125, -0.013708, 3.141563, 0.000000]),accel_mss,speed_ms,0,0.001)
      movel(pose_trans(ref_frame,p[0.113341, 0.114155, -0.000125, -0.013708, 3.141563, -0.000000]),accel_mss,speed_ms,0,0.001)
      movel(pose_trans(ref_frame,p[0.112978, 0.113715, -0.000125, -0.013708, 3.141563, 0.000000]),accel_mss,speed_ms,0,0.001)
      movel(pose_trans(ref_frame,p[0.112537, 0.113377, -0.000125, -0.013708, 3.141563, 0.000000]),accel_mss,speed_ms,0,0.001)
      movel(pose_trans(ref_frame,p[0.112028, 0.113153, -0.000125, -0.013708, 3.141563, 0.000000]),accel_mss,speed_ms,0,0.001)
      movel(pose_trans(ref_frame,p[0.111511, 0.113066, -0.000125, -0.013708, 3.141563, -0.000000]),accel_mss,speed_ms,0,0.001)
      movel(pose_trans(ref_frame,p[0.110988, 0.113113, -0.000125, -0.013708, 3.141563, -0.000000]),accel_mss,speed_ms,0,0.001)
      movel(pose_trans(ref_frame,p[0.110512, 0.113292, -0.000125, -0.013708, 3.141563, 0.000000]),accel_mss,speed_ms,0,0.001)
      movel(pose_trans(ref_frame,p[0.110106, 0.113597, -0.000125, -0.013708, 3.141563, 0.000000]),accel_mss,speed_ms,0,0.001)
      movel(pose_trans(ref_frame,p[0.109649, 0.114258, -0.000125, -0.013708, 3.141563, 0.000000]),accel_mss,speed_ms,0,0.001)
      movel(pose_trans(ref_frame,p[0.109457, 0.115039, -0.000125, -0.013708, 3.141563, 0.000000]),accel_mss,speed_ms,0,0.001)
      movel(pose_trans(ref_frame,p[0.109513, 0.115961, -0.000125, -0.013708, 3.141563, 0.000000]),accel_mss,speed_ms,0,0.001)
      movel(pose_trans(ref_frame,p[0.109788, 0.116843, -0.000125, -0.013708, 3.141563, 0.000000]),accel_mss,speed_ms,0,0.001)
      movel(pose_trans(ref_frame,p[0.110360, 0.117859, -0.000125, -0.013708, 3.141563, 0.000000]),accel_mss,speed_ms,0,0.001)
      movel(pose_trans(ref_frame,p[0.111101, 0.118759, -0.000125, -0.013708, 3.141563, 0.000000]),accel_mss,speed_ms,0,0.001)
      movel(pose_trans(ref_frame,p[0.112108, 0.119673, -0.000125, -0.013708, 3.141563, -0.000000]),accel_mss,speed_ms,0,0.001)
      movel(pose_trans(ref_frame,p[0.113211, 0.120470, -0.000125, -0.013708, 3.141563, 0.000000]),accel_mss,speed_ms,0,0) # end trace
      speed_ms    = 1.000
      movel(pose_trans(ref_frame,p[0.113210, 0.120470, 0.005000, -0.013708, 3.141563, -0.000000]),accel_mss,speed_ms,0,0.001)
      movel(pose_trans(ref_frame,p[0.125304, 0.129232, 0.005000, -0.013708, 3.141563, 0.000000]),accel_mss,speed_ms,0,0) # end trace
      speed_ms    = 0.002
      movel(pose_trans(ref_frame,p[0.125304, 0.129232, -0.000125, -0.013708, 3.141563, 0.000000]),accel_mss,speed_ms,0,0) # end trace
      speed_ms    = 0.007
      movel(pose_trans(ref_frame,p[0.125788, 0.128732, -0.000125, -0.013708, 3.141563, 0.000000]),accel_mss,speed_ms,0,0.001)
      movel(pose_trans(ref_frame,p[0.126269, 0.128230, -0.000125, -0.013708, 3.141563, -0.000000]),accel_mss,speed_ms,0,0.001)
      movel(pose_trans(ref_frame,p[0.126438, 0.128045, -0.000125, -0.013708, 3.141563, -0.000000]),accel_mss,speed_ms,0,0.001)
      movel(pose_trans(ref_frame,p[0.126596, 0.127852, -0.000125, -0.013708, 3.141563, 0.000000]),accel_mss,speed_ms,0,0.001)
      movel(pose_trans(ref_frame,p[0.126662, 0.127750, -0.000125, -0.013708, 3.141563, 0.000000]),accel_mss,speed_ms,0,0.001)
      movel(pose_trans(ref_frame,p[0.126707, 0.127637, -0.000125, -0.013708, 3.141563, -0.000000]),accel_mss,speed_ms,0,0.001)
      movel(pose_trans(ref_frame,p[0.126708, 0.127555, -0.000125, -0.013708, 3.141563, 0.000000]),accel_mss,speed_ms,0,0.001)
      movel(pose_trans(ref_frame,p[0.126668, 0.127483, -0.000125, -0.013708, 3.141563, 0.000000]),accel_mss,speed_ms,0,0.001)
      movel(pose_trans(ref_frame,p[0.126614, 0.127443, -0.000125, -0.013708, 3.141563, -0.000000]),accel_mss,speed_ms,0,0.001)
      movel(pose_trans(ref_frame,p[0.126552, 0.127419, -0.000125, -0.013708, 3.141563, 0.000000]),accel_mss,speed_ms,0,0.001)
      movel(pose_trans(ref_frame,p[0.126476, 0.127409, -0.000125, -0.013708, 3.141563, 0.000000]),accel_mss,speed_ms,0,0.001)
      movel(pose_trans(ref_frame,p[0.126399, 0.127414, -0.000125, -0.013708, 3.141563, -0.000000]),accel_mss,speed_ms,0,0.001)
      movel(pose_trans(ref_frame,p[0.126292, 0.127437, -0.000125, -0.013708, 3.141563, -0.000000]),accel_mss,speed_ms,0,0.001)
      movel(pose_trans(ref_frame,p[0.126187, 0.127472, -0.000125, -0.013708, 3.141563, 0.000000]),accel_mss,speed_ms,0,0.001)
      movel(pose_trans(ref_frame,p[0.126030, 0.127537, -0.000125, -0.013708, 3.141563, 0.000000]),accel_mss,speed_ms,0,0.001)
      movel(pose_trans(ref_frame,p[0.125875, 0.127607, -0.000125, -0.013708, 3.141563, 0.000000]),accel_mss,speed_ms,0,0.001)
      movel(pose_trans(ref_frame,p[0.125369, 0.127792, -0.000125, -0.013708, 3.141563, 0.000000]),accel_mss,speed_ms,0,0.001)
      movel(pose_trans(ref_frame,p[0.124838, 0.127884, -0.000125, -0.013708, 3.141563, -0.000000]),accel_mss,speed_ms,0,0.001)
      movel(pose_trans(ref_frame,p[0.124236, 0.127895, -0.000125, -0.013708, 3.141563, 0.000000]),accel_mss,speed_ms,0,0.001)
      movel(pose_trans(ref_frame,p[0.123638, 0.127828, -0.000125, -0.013708, 3.141563, 0.000000]),accel_mss,speed_ms,0,0.001)
      movel(pose_trans(ref_frame,p[0.123019, 0.127679, -0.000125, -0.013708, 3.141563, -0.000000]),accel_mss,speed_ms,0,0.001)
      movel(pose_trans(ref_frame,p[0.122422, 0.127455, -0.000125, -0.013708, 3.141563, 0.000000]),accel_mss,speed_ms,0,0.001)
      movel(pose_trans(ref_frame,p[0.121859, 0.127161, -0.000125, -0.013708, 3.141563, -0.000000]),accel_mss,speed_ms,0,0.001)
      movel(pose_trans(ref_frame,p[0.121335, 0.126800, -0.000125, -0.013708, 3.141563, 0.000000]),accel_mss,speed_ms,0,0.001)
      movel(pose_trans(ref_frame,p[0.120642, 0.126257, -0.000125, -0.013708, 3.141563, -0.000000]),accel_mss,speed_ms,0,0.001)
      movel(pose_trans(ref_frame,p[0.121900, 0.124999, -0.000125, -0.013708, 3.141563, 0.000000]),accel_mss,speed_ms,0,0.001)
      movel(pose_trans(ref_frame,p[0.123158, 0.123741, -0.000125, -0.013708, 3.141563, -0.000000]),accel_mss,speed_ms,0,0.001)
      movel(pose_trans(ref_frame,p[0.123706, 0.124174, -0.000125, -0.013708, 3.141563, -0.000000]),accel_mss,speed_ms,0,0.001)
      movel(pose_trans(ref_frame,p[0.124584, 0.124819, -0.000125, -0.013708, 3.141563, -0.000000]),accel_mss,speed_ms,0,0.001)
      movel(pose_trans(ref_frame,p[0.125505, 0.125401, -0.000125, -0.013708, 3.141563, 0.000000]),accel_mss,speed_ms,0,0.001)
      movel(pose_trans(ref_frame,p[0.126317, 0.125813, -0.000125, -0.013708, 3.141563, 0.000000]),accel_mss,speed_ms,0,0.001)
      movel(pose_trans(ref_frame,p[0.127172, 0.126128, -0.000125, -0.013708, 3.141563, 0.000000]),accel_mss,speed_ms,0,0.001)
      movel(pose_trans(ref_frame,p[0.127935, 0.126300, -0.000125, -0.013708, 3.141563, 0.000000]),accel_mss,speed_ms,0,0.001)
      movel(pose_trans(ref_frame,p[0.128714, 0.126361, -0.000125, -0.013708, 3.141563, -0.000000]),accel_mss,speed_ms,0,0.001)
      movel(pose_trans(ref_frame,p[0.129435, 0.126302, -0.000125, -0.013708, 3.141563, -0.000000]),accel_mss,speed_ms,0,0.001)
      movel(pose_trans(ref_frame,p[0.130135, 0.126116, -0.000125, -0.013708, 3.141563, 0.000000]),accel_mss,speed_ms,0,0.001)
      movel(pose_trans(ref_frame,p[0.130337, 0.126037, -0.000125, -0.013708, 3.141563, 0.000000]),accel_mss,speed_ms,0,0.001)
      movel(pose_trans(ref_frame,p[0.130534, 0.125949, -0.000125, -0.013708, 3.141563, -0.000000]),accel_mss,speed_ms,0,0.001)
      movel(pose_trans(ref_frame,p[0.130693, 0.125866, -0.000125, -0.013708, 3.141563, -0.000000]),accel_mss,speed_ms,0,0.001)
      movel(pose_trans(ref_frame,p[0.130845, 0.125770, -0.000125, -0.013708, 3.141563, 0.000000]),accel_mss,speed_ms,0,0.001)
      movel(pose_trans(ref_frame,p[0.131005, 0.125652, -0.000125, -0.013708, 3.141563, -0.000000]),accel_mss,speed_ms,0,0.001)
      movel(pose_trans(ref_frame,p[0.131156, 0.125524, -0.000125, -0.013708, 3.141563, 0.000000]),accel_mss,speed_ms,0,0.001)
      movel(pose_trans(ref_frame,p[0.131364, 0.125331, -0.000125, -0.013708, 3.141563, -0.000000]),accel_mss,speed_ms,0,0.001)
      movel(pose_trans(ref_frame,p[0.131567, 0.125133, -0.000125, -0.013708, 3.141563, -0.000000]),accel_mss,speed_ms,0,0.001)
      movel(pose_trans(ref_frame,p[0.131767, 0.124927, -0.000125, -0.013708, 3.141563, 0.000000]),accel_mss,speed_ms,0,0.001)
      movel(pose_trans(ref_frame,p[0.131963, 0.124717, -0.000125, -0.013708, 3.141563, 0.000000]),accel_mss,speed_ms,0,0.001)
      movel(pose_trans(ref_frame,p[0.132091, 0.124564, -0.000125, -0.013708, 3.141563, 0.000000]),accel_mss,speed_ms,0,0.001)
      movel(pose_trans(ref_frame,p[0.132209, 0.124404, -0.000125, -0.013708, 3.141563, 0.000000]),accel_mss,speed_ms,0,0.001)
      movel(pose_trans(ref_frame,p[0.132306, 0.124248, -0.000125, -0.013708, 3.141563, 0.000000]),accel_mss,speed_ms,0,0.001)
      movel(pose_trans(ref_frame,p[0.132390, 0.124084, -0.000125, -0.013708, 3.141563, 0.000000]),accel_mss,speed_ms,0,0.001)
      movel(pose_trans(ref_frame,p[0.132483, 0.123874, -0.000125, -0.013708, 3.141563, -0.000000]),accel_mss,speed_ms,0,0.001)
      movel(pose_trans(ref_frame,p[0.132567, 0.123660, -0.000125, -0.013708, 3.141563, -0.000000]),accel_mss,speed_ms,0,0.001)
      movel(pose_trans(ref_frame,p[0.132817, 0.122543, -0.000125, -0.013708, 3.141563, 0.000000]),accel_mss,speed_ms,0,0.001)
      movel(pose_trans(ref_frame,p[0.132765, 0.121400, -0.000125, -0.013708, 3.141563, -0.000000]),accel_mss,speed_ms,0,0.001)
      movel(pose_trans(ref_frame,p[0.132421, 0.120115, -0.000125, -0.013708, 3.141563, 0.000000]),accel_mss,speed_ms,0,0.001)
      movel(pose_trans(ref_frame,p[0.131863, 0.118908, -0.000125, -0.013708, 3.141563, 0.000000]),accel_mss,speed_ms,0,0.001)
      movel(pose_trans(ref_frame,p[0.131071, 0.117744, -0.000125, -0.013708, 3.141563, -0.000000]),accel_mss,speed_ms,0,0.001)
      movel(pose_trans(ref_frame,p[0.130103, 0.116721, -0.000125, -0.013708, 3.141563, 0.000000]),accel_mss,speed_ms,0,0.001)
      movel(pose_trans(ref_frame,p[0.129032, 0.115926, -0.000125, -0.013708, 3.141563, -0.000000]),accel_mss,speed_ms,0,0.001)
      movel(pose_trans(ref_frame,p[0.127831, 0.115345, -0.000125, -0.013708, 3.141563, 0.000000]),accel_mss,speed_ms,0,0.001)
      movel(pose_trans(ref_frame,p[0.127388, 0.115203, -0.000125, -0.013708, 3.141563, 0.000000]),accel_mss,speed_ms,0,0.001)
      movel(pose_trans(ref_frame,p[0.126934, 0.115104, -0.000125, -0.013708, 3.141563, -0.000000]),accel_mss,speed_ms,0,0.001)
      movel(pose_trans(ref_frame,p[0.126538, 0.115066, -0.000125, -0.013708, 3.141563, 0.000000]),accel_mss,speed_ms,0,0.001)
      movel(pose_trans(ref_frame,p[0.126141, 0.115089, -0.000125, -0.013708, 3.141563, -0.000000]),accel_mss,speed_ms,0,0.001)
      movel(pose_trans(ref_frame,p[0.125786, 0.115167, -0.000125, -0.013708, 3.141563, -0.000000]),accel_mss,speed_ms,0,0.001)
      movel(pose_trans(ref_frame,p[0.125449, 0.115304, -0.000125, -0.013708, 3.141563, 0.000000]),accel_mss,speed_ms,0,0.001)
      movel(pose_trans(ref_frame,p[0.125132, 0.115498, -0.000125, -0.013708, 3.141563, 0.000000]),accel_mss,speed_ms,0,0.001)
      movel(pose_trans(ref_frame,p[0.124848, 0.115740, -0.000125, -0.013708, 3.141563, 0.000000]),accel_mss,speed_ms,0,0.001)
      movel(pose_trans(ref_frame,p[0.124622, 0.116015, -0.000125, -0.013708, 3.141563, 0.000000]),accel_mss,speed_ms,0,0.001)
      movel(pose_trans(ref_frame,p[0.124452, 0.116327, -0.000125, -0.013708, 3.141563, 0.000000]),accel_mss,speed_ms,0,0.001)
      movel(pose_trans(ref_frame,p[0.124350, 0.116660, -0.000125, -0.013708, 3.141563, 0.000000]),accel_mss,speed_ms,0,0.001)
      movel(pose_trans(ref_frame,p[0.124319, 0.117006, -0.000125, -0.013708, 3.141563, -0.000000]),accel_mss,speed_ms,0,0.001)
      movel(pose_trans(ref_frame,p[0.124358, 0.117369, -0.000125, -0.013708, 3.141563, -0.000000]),accel_mss,speed_ms,0,0.001)
      movel(pose_trans(ref_frame,p[0.124466, 0.117717, -0.000125, -0.013708, 3.141563, -0.000000]),accel_mss,speed_ms,0,0.001)
      movel(pose_trans(ref_frame,p[0.124648, 0.118072, -0.000125, -0.013708, 3.141563, -0.000000]),accel_mss,speed_ms,0,0.001)
      movel(pose_trans(ref_frame,p[0.124880, 0.118397, -0.000125, -0.013708, 3.141563, 0.000000]),accel_mss,speed_ms,0,0.001)
      movel(pose_trans(ref_frame,p[0.125096, 0.118629, -0.000125, -0.013708, 3.141563, 0.000000]),accel_mss,speed_ms,0,0.001)
      movel(pose_trans(ref_frame,p[0.125335, 0.118837, -0.000125, -0.013708, 3.141563, -0.000000]),accel_mss,speed_ms,0,0.001)
      movel(pose_trans(ref_frame,p[0.125578, 0.119002, -0.000125, -0.013708, 3.141563, -0.000000]),accel_mss,speed_ms,0,0.001)
      movel(pose_trans(ref_frame,p[0.125841, 0.119133, -0.000125, -0.013708, 3.141563, -0.000000]),accel_mss,speed_ms,0,0.001)
      movel(pose_trans(ref_frame,p[0.126105, 0.119221, -0.000125, -0.013708, 3.141563, -0.000000]),accel_mss,speed_ms,0,0.001)
      movel(pose_trans(ref_frame,p[0.126379, 0.119271, -0.000125, -0.013708, 3.141563, 0.000000]),accel_mss,speed_ms,0,0.001)
      movel(pose_trans(ref_frame,p[0.126654, 0.119280, -0.000125, -0.013708, 3.141563, 0.000000]),accel_mss,speed_ms,0,0.001)
      movel(pose_trans(ref_frame,p[0.126926, 0.119248, -0.000125, -0.013708, 3.141563, 0.000000]),accel_mss,speed_ms,0,0.001)
      movel(pose_trans(ref_frame,p[0.127168, 0.119178, -0.000125, -0.013708, 3.141563, 0.000000]),accel_mss,speed_ms,0,0.001)
      movel(pose_trans(ref_frame,p[0.127394, 0.119067, -0.000125, -0.013708, 3.141563, 0.000000]),accel_mss,speed_ms,0,0.001)
      movel(pose_trans(ref_frame,p[0.127636, 0.118900, -0.000125, -0.013708, 3.141563, -0.000000]),accel_mss,speed_ms,0,0.001)
      movel(pose_trans(ref_frame,p[0.127859, 0.118707, -0.000125, -0.013708, 3.141563, 0.000000]),accel_mss,speed_ms,0,0.001)
      movel(pose_trans(ref_frame,p[0.128064, 0.118485, -0.000125, -0.013708, 3.141563, 0.000000]),accel_mss,speed_ms,0,0.001)
      movel(pose_trans(ref_frame,p[0.128245, 0.118241, -0.000125, -0.013708, 3.141563, 0.000000]),accel_mss,speed_ms,0,0.001)
      movel(pose_trans(ref_frame,p[0.128380, 0.118000, -0.000125, -0.013708, 3.141563, -0.000000]),accel_mss,speed_ms,0,0.001)
      movel(pose_trans(ref_frame,p[0.128478, 0.117742, -0.000125, -0.013708, 3.141563, -0.000000]),accel_mss,speed_ms,0,0.001)
      movel(pose_trans(ref_frame,p[0.128624, 0.117258, -0.000125, -0.013708, 3.141563, 0.000000]),accel_mss,speed_ms,0,0.001)
      movel(pose_trans(ref_frame,p[0.128944, 0.117315, -0.000125, -0.013708, 3.141563, 0.000000]),accel_mss,speed_ms,0,0.001)
      movel(pose_trans(ref_frame,p[0.129262, 0.117427, -0.000125, -0.013708, 3.141563, 0.000000]),accel_mss,speed_ms,0,0.001)
      movel(pose_trans(ref_frame,p[0.129526, 0.117636, -0.000125, -0.013708, 3.141563, -0.000000]),accel_mss,speed_ms,0,0.001)
      movel(pose_trans(ref_frame,p[0.129760, 0.117956, -0.000125, -0.013708, 3.141563, 0.000000]),accel_mss,speed_ms,0,0.001)
      movel(pose_trans(ref_frame,p[0.129923, 0.118316, -0.000125, -0.013708, 3.141563, -0.000000]),accel_mss,speed_ms,0,0.001)
      movel(pose_trans(ref_frame,p[0.130027, 0.118756, -0.000125, -0.013708, 3.141563, 0.000000]),accel_mss,speed_ms,0,0.001)
      movel(pose_trans(ref_frame,p[0.130053, 0.119207, -0.000125, -0.013708, 3.141563, 0.000000]),accel_mss,speed_ms,0,0.001)
      movel(pose_trans(ref_frame,p[0.130001, 0.119668, -0.000125, -0.013708, 3.141563, 0.000000]),accel_mss,speed_ms,0,0.001)
      movel(pose_trans(ref_frame,p[0.129875, 0.120115, -0.000125, -0.013708, 3.141563, 0.000000]),accel_mss,speed_ms,0,0.001)
      movel(pose_trans(ref_frame,p[0.129735, 0.120423, -0.000125, -0.013708, 3.141563, -0.000000]),accel_mss,speed_ms,0,0.001)
      movel(pose_trans(ref_frame,p[0.129552, 0.120707, -0.000125, -0.013708, 3.141563, 0.000000]),accel_mss,speed_ms,0,0.001)
      movel(pose_trans(ref_frame,p[0.129297, 0.121019, -0.000125, -0.013708, 3.141563, 0.000000]),accel_mss,speed_ms,0,0.001)
      movel(pose_trans(ref_frame,p[0.129015, 0.121309, -0.000125, -0.013708, 3.141563, 0.000000]),accel_mss,speed_ms,0,0.001)
      movel(pose_trans(ref_frame,p[0.128708, 0.121576, -0.000125, -0.013708, 3.141563, 0.000000]),accel_mss,speed_ms,0,0.001)
      movel(pose_trans(ref_frame,p[0.128378, 0.121816, -0.000125, -0.013708, 3.141563, 0.000000]),accel_mss,speed_ms,0,0.001)
      movel(pose_trans(ref_frame,p[0.128074, 0.121991, -0.000125, -0.013708, 3.141563, 0.000000]),accel_mss,speed_ms,0,0.001)
      movel(pose_trans(ref_frame,p[0.127750, 0.122124, -0.000125, -0.013708, 3.141563, -0.000000]),accel_mss,speed_ms,0,0.001)
      movel(pose_trans(ref_frame,p[0.127455, 0.122208, -0.000125, -0.013708, 3.141563, 0.000000]),accel_mss,speed_ms,0,0.001)
      movel(pose_trans(ref_frame,p[0.127153, 0.122265, -0.000125, -0.013708, 3.141563, 0.000000]),accel_mss,speed_ms,0,0.001)
      movel(pose_trans(ref_frame,p[0.126835, 0.122297, -0.000125, -0.013708, 3.141563, -0.000000]),accel_mss,speed_ms,0,0.001)
      movel(pose_trans(ref_frame,p[0.126515, 0.122304, -0.000125, -0.013708, 3.141563, 0.000000]),accel_mss,speed_ms,0,0.001)
      movel(pose_trans(ref_frame,p[0.126184, 0.122284, -0.000125, -0.013708, 3.141563, 0.000000]),accel_mss,speed_ms,0,0.001)
      movel(pose_trans(ref_frame,p[0.125855, 0.122238, -0.000125, -0.013708, 3.141563, 0.000000]),accel_mss,speed_ms,0,0.001)
      movel(pose_trans(ref_frame,p[0.125519, 0.122166, -0.000125, -0.013708, 3.141563, -0.000000]),accel_mss,speed_ms,0,0.001)
      movel(pose_trans(ref_frame,p[0.125189, 0.122071, -0.000125, -0.013708, 3.141563, 0.000000]),accel_mss,speed_ms,0,0.001)
      movel(pose_trans(ref_frame,p[0.124895, 0.121966, -0.000125, -0.013708, 3.141563, -0.000000]),accel_mss,speed_ms,0,0.001)
      movel(pose_trans(ref_frame,p[0.124607, 0.121845, -0.000125, -0.013708, 3.141563, -0.000000]),accel_mss,speed_ms,0,0.001)
      movel(pose_trans(ref_frame,p[0.124339, 0.121713, -0.000125, -0.013708, 3.141563, 0.000000]),accel_mss,speed_ms,0,0.001)
      movel(pose_trans(ref_frame,p[0.124079, 0.121565, -0.000125, -0.013708, 3.141563, 0.000000]),accel_mss,speed_ms,0,0.001)
      movel(pose_trans(ref_frame,p[0.123788, 0.121377, -0.000125, -0.013708, 3.141563, 0.000000]),accel_mss,speed_ms,0,0.001)
      movel(pose_trans(ref_frame,p[0.123507, 0.121175, -0.000125, -0.013708, 3.141563, 0.000000]),accel_mss,speed_ms,0,0.001)
      movel(pose_trans(ref_frame,p[0.123138, 0.120889, -0.000125, -0.013708, 3.141563, 0.000000]),accel_mss,speed_ms,0,0.001)
      movel(pose_trans(ref_frame,p[0.122776, 0.120595, -0.000125, -0.013708, 3.141563, 0.000000]),accel_mss,speed_ms,0,0.001)
      movel(pose_trans(ref_frame,p[0.122607, 0.120457, -0.000125, -0.013708, 3.141563, -0.000000]),accel_mss,speed_ms,0,0.001)
      movel(pose_trans(ref_frame,p[0.122437, 0.120321, -0.000125, -0.013708, 3.141563, -0.000000]),accel_mss,speed_ms,0,0.001)
      movel(pose_trans(ref_frame,p[0.122283, 0.120201, -0.000125, -0.013708, 3.141563, 0.000000]),accel_mss,speed_ms,0,0.001)
      movel(pose_trans(ref_frame,p[0.122127, 0.120084, -0.000125, -0.013708, 3.141563, 0.000000]),accel_mss,speed_ms,0,0.001)
      movel(pose_trans(ref_frame,p[0.121996, 0.119987, -0.000125, -0.013708, 3.141563, 0.000000]),accel_mss,speed_ms,0,0.001)
      movel(pose_trans(ref_frame,p[0.121863, 0.119892, -0.000125, -0.013708, 3.141563, 0.000000]),accel_mss,speed_ms,0,0.001)
      movel(pose_trans(ref_frame,p[0.121819, 0.119867, -0.000125, -0.013708, 3.141563, 0.000000]),accel_mss,speed_ms,0,0.001)
      movel(pose_trans(ref_frame,p[0.121772, 0.119851, -0.000125, -0.013708, 3.141563, -0.000000]),accel_mss,speed_ms,0,0.001)
      movel(pose_trans(ref_frame,p[0.121663, 0.119853, -0.000125, -0.013708, 3.141563, -0.000000]),accel_mss,speed_ms,0,0.001)
      movel(pose_trans(ref_frame,p[0.121569, 0.119907, -0.000125, -0.013708, 3.141563, -0.000000]),accel_mss,speed_ms,0,0.001)
      movel(pose_trans(ref_frame,p[0.120525, 0.120931, -0.000125, -0.013708, 3.141563, 0.000000]),accel_mss,speed_ms,0,0.001)
      movel(pose_trans(ref_frame,p[0.119482, 0.121957, -0.000125, -0.013708, 3.141563, 0.000000]),accel_mss,speed_ms,0,0.001)
      movel(pose_trans(ref_frame,p[0.118447, 0.122978, -0.000125, -0.013708, 3.141563, -0.000000]),accel_mss,speed_ms,0,0.001)
      movel(pose_trans(ref_frame,p[0.117414, 0.124000, -0.000125, -0.013708, 3.141563, 0.000000]),accel_mss,speed_ms,0,0.001)
      movel(pose_trans(ref_frame,p[0.117340, 0.124110, -0.000125, -0.013708, 3.141563, 0.000000]),accel_mss,speed_ms,0,0.001)
      movel(pose_trans(ref_frame,p[0.117314, 0.124241, -0.000125, -0.013708, 3.141563, 0.000000]),accel_mss,speed_ms,0,0.001)
      movel(pose_trans(ref_frame,p[0.117322, 0.124283, -0.000125, -0.013708, 3.141563, 0.000000]),accel_mss,speed_ms,0,0.001)
      movel(pose_trans(ref_frame,p[0.117345, 0.124319, -0.000125, -0.013708, 3.141563, -0.000000]),accel_mss,speed_ms,0,0.001)
      movel(pose_trans(ref_frame,p[0.117803, 0.124794, -0.000125, -0.013708, 3.141563, -0.000000]),accel_mss,speed_ms,0,0.001)
      movel(pose_trans(ref_frame,p[0.118262, 0.125270, -0.000125, -0.013708, 3.141563, 0.000000]),accel_mss,speed_ms,0,0.001)
      movel(pose_trans(ref_frame,p[0.118782, 0.125805, -0.000125, -0.013708, 3.141563, -0.000000]),accel_mss,speed_ms,0,0.001)
      movel(pose_trans(ref_frame,p[0.119304, 0.126337, -0.000125, -0.013708, 3.141563, 0.000000]),accel_mss,speed_ms,0,0.001)
      movel(pose_trans(ref_frame,p[0.119922, 0.126961, -0.000125, -0.013708, 3.141563, -0.000000]),accel_mss,speed_ms,0,0.001)
      movel(pose_trans(ref_frame,p[0.120542, 0.127583, -0.000125, -0.013708, 3.141563, -0.000000]),accel_mss,speed_ms,0,0.001)
      movel(pose_trans(ref_frame,p[0.123771, 0.130812, -0.000125, -0.013708, 3.141563, 0.000000]),accel_mss,speed_ms,0,0.001)
      movel(pose_trans(ref_frame,p[0.125304, 0.129232, -0.000125, -0.013708, 3.141563, 0.000000]),accel_mss,speed_ms,0,0) # end trace
      speed_ms    = 1.000
      movel(pose_trans(ref_frame,p[0.125304, 0.129232, 0.005000, -0.013708, 3.141563, 0.000000]),accel_mss,speed_ms,0,0.001)
      movel(pose_trans(ref_frame,p[0.016011, 0.134006, 0.005000, -0.013708, 3.141563, 0.000000]),accel_mss,speed_ms,0,0) # end trace
      speed_ms    = 0.002
      movel(pose_trans(ref_frame,p[0.016011, 0.134006, -0.000125, -0.013708, 3.141563, 0.000000]),accel_mss,speed_ms,0,0) # end trace
      speed_ms    = 0.007
      movel(pose_trans(ref_frame,p[0.016016, 0.132903, -0.000125, -0.013708, 3.141563, 0.000000]),accel_mss,speed_ms,0,0.001)
      movel(pose_trans(ref_frame,p[0.016912, 0.132897, -0.000125, -0.013708, 3.141563, -0.000000]),accel_mss,speed_ms,0,0.001)
      movel(pose_trans(ref_frame,p[0.017086, 0.132895, -0.000125, -0.013708, 3.141563, 0.000000]),accel_mss,speed_ms,0,0.001)
      movel(pose_trans(ref_frame,p[0.017260, 0.132891, -0.000125, -0.013708, 3.141563, -0.000000]),accel_mss,speed_ms,0,0.001)
      movel(pose_trans(ref_frame,p[0.017411, 0.132885, -0.000125, -0.013708, 3.141563, -0.000000]),accel_mss,speed_ms,0,0.001)
      movel(pose_trans(ref_frame,p[0.017562, 0.132876, -0.000125, -0.013708, 3.141563, -0.000000]),accel_mss,speed_ms,0,0.001)
      movel(pose_trans(ref_frame,p[0.017689, 0.132866, -0.000125, -0.013708, 3.141563, -0.000000]),accel_mss,speed_ms,0,0.001)
      movel(pose_trans(ref_frame,p[0.017816, 0.132855, -0.000125, -0.013708, 3.141563, 0.000000]),accel_mss,speed_ms,0,0.001)
      movel(pose_trans(ref_frame,p[0.017844, 0.132848, -0.000125, -0.013708, 3.141563, 0.000000]),accel_mss,speed_ms,0,0.001)
      movel(pose_trans(ref_frame,p[0.017869, 0.132831, -0.000125, -0.013708, 3.141563, 0.000000]),accel_mss,speed_ms,0,0.001)
      movel(pose_trans(ref_frame,p[0.017926, 0.132747, -0.000125, -0.013708, 3.141563, 0.000000]),accel_mss,speed_ms,0,0.001)
      movel(pose_trans(ref_frame,p[0.017949, 0.132648, -0.000125, -0.013708, 3.141563, 0.000000]),accel_mss,speed_ms,0,0.001)
      movel(pose_trans(ref_frame,p[0.017959, 0.132366, -0.000125, -0.013708, 3.141563, 0.000000]),accel_mss,speed_ms,0,0.001)
      movel(pose_trans(ref_frame,p[0.017961, 0.132083, -0.000125, -0.013708, 3.141563, 0.000000]),accel_mss,speed_ms,0,0.001)
      movel(pose_trans(ref_frame,p[0.017955, 0.131800, -0.000125, -0.013708, 3.141563, 0.000000]),accel_mss,speed_ms,0,0.001)
      movel(pose_trans(ref_frame,p[0.017942, 0.131518, -0.000125, -0.013708, 3.141563, 0.000000]),accel_mss,speed_ms,0,0.001)
      movel(pose_trans(ref_frame,p[0.017917, 0.131418, -0.000125, -0.013708, 3.141563, -0.000000]),accel_mss,speed_ms,0,0.001)
      movel(pose_trans(ref_frame,p[0.017859, 0.131334, -0.000125, -0.013708, 3.141563, 0.000000]),accel_mss,speed_ms,0,0.001)
      movel(pose_trans(ref_frame,p[0.017813, 0.131300, -0.000125, -0.013708, 3.141563, -0.000000]),accel_mss,speed_ms,0,0.001)
      movel(pose_trans(ref_frame,p[0.017760, 0.131280, -0.000125, -0.013708, 3.141563, 0.000000]),accel_mss,speed_ms,0,0.001)
      movel(pose_trans(ref_frame,p[0.017636, 0.131256, -0.000125, -0.013708, 3.141563, 0.000000]),accel_mss,speed_ms,0,0.001)
      movel(pose_trans(ref_frame,p[0.017510, 0.131235, -0.000125, -0.013708, 3.141563, 0.000000]),accel_mss,speed_ms,0,0.001)
      movel(pose_trans(ref_frame,p[0.017357, 0.131217, -0.000125, -0.013708, 3.141563, -0.000000]),accel_mss,speed_ms,0,0.001)
      movel(pose_trans(ref_frame,p[0.017203, 0.131204, -0.000125, -0.013708, 3.141563, 0.000000]),accel_mss,speed_ms,0,0.001)
      movel(pose_trans(ref_frame,p[0.017034, 0.131195, -0.000125, -0.013708, 3.141563, -0.000000]),accel_mss,speed_ms,0,0.001)
      movel(pose_trans(ref_frame,p[0.016864, 0.131192, -0.000125, -0.013708, 3.141563, 0.000000]),accel_mss,speed_ms,0,0.001)
      movel(pose_trans(ref_frame,p[0.016006, 0.131186, -0.000125, -0.013708, 3.141563, 0.000000]),accel_mss,speed_ms,0,0.001)
      movel(pose_trans(ref_frame,p[0.016011, 0.130119, -0.000125, -0.013708, 3.141563, -0.000000]),accel_mss,speed_ms,0,0.001)
      movel(pose_trans(ref_frame,p[0.016016, 0.129053, -0.000125, -0.013708, 3.141563, -0.000000]),accel_mss,speed_ms,0,0.001)
      movel(pose_trans(ref_frame,p[0.017074, 0.129051, -0.000125, -0.013708, 3.141563, -0.000000]),accel_mss,speed_ms,0,0.001)
      movel(pose_trans(ref_frame,p[0.017279, 0.129052, -0.000125, -0.013708, 3.141563, 0.000000]),accel_mss,speed_ms,0,0.001)
      movel(pose_trans(ref_frame,p[0.017484, 0.129054, -0.000125, -0.013708, 3.141563, 0.000000]),accel_mss,speed_ms,0,0.001)
      movel(pose_trans(ref_frame,p[0.017661, 0.129058, -0.000125, -0.013708, 3.141563, -0.000000]),accel_mss,speed_ms,0,0.001)
      movel(pose_trans(ref_frame,p[0.017837, 0.129065, -0.000125, -0.013708, 3.141563, 0.000000]),accel_mss,speed_ms,0,0.001)
